LIN {X 0,Y 360.058,Z 331.263,A -85,B 0,C 180,E1 -13391.69,E2 -13391.69} C_VEL
LIN {X 0,Y 358.876,Z 343.094,A -85,B 0,C 180,E1 -13392.772,E2 -13392.772} C_VEL
LIN {X 0,Y 357.607,Z 353.882,A -85,B 0,C 180,E1 -13394.031,E2 -13394.031} C_VEL
LIN {X 0,Y 356.56,Z 363.612,A -85,B 0,C 180,E1 -13395.447,E2 -13395.447} C_VEL
LIN {X 0,Y 355.69,Z 371.607,A -85,B 0,C 180,E1 -13396.868,E2 -13396.868} C_VEL
LIN {X 0,Y 354.707,Z 379.453,A -85,B 0,C 180,E1 -13398.574,E2 -13398.574} C_VEL
LIN {X 0,Y 354.087,Z 385.752,A -85,B 0,C 180,E1 -13400.289,E2 -13400.289} C_VEL
LIN {X 0,Y 353.652,Z 390.778,A -85,B 0,C 180,E1 -13402.005,E2 -13402.005} C_VEL
LIN {X 0,Y 353.422,Z 394.956,A -85,B 0,C 180,E1 -13403.87,E2 -13403.87} C_VEL
LIN {X 0,Y 353.356,Z 397.554,A -85,B 0,C 180,E1 -13405.439,E2 -13405.439} C_VEL
LIN {X 0,Y 353.303,Z 399.885,A -85,B 0,C 180,E1 -13407.722,E2 -13407.722} C_VEL
LIN {X 0,Y 353.398,Z 400.466,A -85,B 0,C 180,E1 -13408.862,E2 -13408.862} C_VEL
LIN {X 0,Y 353.411,Z 400.609,A -85,B 0,C 180,E1 -13410.002,E2 -13410.002} C_VEL
LIN {X 0,Y 353.42,Z 400.345,A -85,B 0,C 180,E1 -13411.141,E2 -13411.141} C_VEL
LIN {X 0,Y 353.334,Z 399.683,A -85,B 0,C 180,E1 -13412.282,E2 -13412.282} C_VEL
LIN {X 0,Y 353.285,Z 398.629,A -85,B 0,C 180,E1 -13413.423,E2 -13413.423} C_VEL
LIN {X 0,Y 353.361,Z 397.134,A -85,B 0,C 180,E1 -13414.565,E2 -13414.565} C_VEL
LIN {X 0,Y 353.448,Z 394.313,A -85,B 0,C 180,E1 -13416.169,E2 -13416.169} C_VEL
LIN {X 0,Y 353.68,Z 389.954,A -85,B 0,C 180,E1 -13417.997,E2 -13417.997} C_VEL
LIN {X 0,Y 354.204,Z 383.631,A -85,B 0,C 180,E1 -13420,E2 -13420} C_VEL
LIN {X 0,Y 354.815,Z 376.746,A -85,B 0,C 180,E1 -13421.716,E2 -13421.716} C_VEL
LIN {X 0,Y 355.758,Z 368.183,A -85,B 0,C 180,E1 -13423.424,E2 -13423.424} C_VEL
LIN {X 0,Y 356.833,Z 358.104,A -85,B 0,C 180,E1 -13425.024,E2 -13425.024} C_VEL
LIN {X 0,Y 357.848,Z 347.306,A -85,B 0,C 180,E1 -13426.4,E2 -13426.4} C_VEL
LIN {X 0,Y 358.984,Z 336.101,A -85,B 0,C 180,E1 -13427.519,E2 -13427.519} C_VEL
LIN {X 0,Y 359.355,Z 329.321,A -85,B 0,C 180,E1 -13428.089,E2 -13428.089} C_VEL
LIN {X 0,Y 358.031,Z 317.342,A -85,B 0,C 180,E1 -13428.993,E2 -13428.993} C_VEL
LIN {X 0,Y 356.267,Z 304.211,A -85,B 0,C 180,E1 -13429.746,E2 -13429.746} C_VEL
LIN {X 0,Y 354.344,Z 292.6,A -85,B 0,C 180,E1 -13430.25,E2 -13430.25} C_VEL
LIN {X 0,Y 354.862,Z 285.094,A -85,B 0,C 180,E1 -13433.858,E2 -13433.858} C_VEL
LIN {X 0,Y 355.458,Z 278.242,A -85,B 0,C 180,E1 -13437.161,E2 -13437.161} C_VEL
LIN {X 0,Y 356.084,Z 272.036,A -85,B 0,C 180,E1 -13440.223,E2 -13440.223} C_VEL
LIN {X 0,Y 356.8,Z 265.53,A -85,B 0,C 180,E1 -13443.473,E2 -13443.473} C_VEL
LIN {X 0,Y 357.286,Z 260.221,A -85,B 0,C 180,E1 -13446.245,E2 -13446.245} C_VEL
LIN {X 0,Y 357.088,Z 256.908,A -85,B 0,C 180,E1 -13448.07,E2 -13448.07} C_VEL
LIN {X 0,Y 356.109,Z 251.252,A -85,B 0,C 180,E1 -13451.414,E2 -13451.414} C_VEL
LIN {X 0,Y 355.185,Z 246.213,A -85,B 0,C 180,E1 -13454.575,E2 -13454.575} C_VEL
LIN {X 0,Y 354.819,Z 244.293,A -85,B 0,C 180,E1 -13455.947,E2 -13455.947} C_VEL
LIN {X 0,Y 354.794,Z 244.292,A -85,B 0,C 180,E1 -13459.18,E2 -13459.18} C_VEL
LIN {X 0,Y 354.813,Z 244.288,A -85,B 0,C 180,E1 -13462.404,E2 -13462.404} C_VEL
LIN {X 0,Y 354.818,Z 244.287,A -85,B 0,C 180,E1 -13464.941,E2 -13464.941} C_VEL
LIN {X 0,Y 354.8,Z 244.292,A -85,B 0,C 180,E1 -13468.406,E2 -13468.406} C_VEL
LIN {X 0,Y 354.817,Z 244.284,A -85,B 0,C 180,E1 -13471.616,E2 -13471.616} C_VEL
LIN {X 0,Y 354.861,Z 244.279,A -85,B 0,C 180,E1 -13475.424,E2 -13475.424} C_VEL
LIN {X 0,Y 354.834,Z 244.282,A -85,B 0,C 180,E1 -13479.114,E2 -13479.114} C_VEL
LIN {X 0,Y 354.867,Z 244.279,A -85,B 0,C 180,E1 -13482.718,E2 -13482.718} C_VEL
LIN {X 0,Y 354.947,Z 244.271,A -85,B 0,C 180,E1 -13486.255,E2 -13486.255} C_VEL
LIN {X 0,Y 354.959,Z 244.272,A -85,B 0,C 180,E1 -13489.735,E2 -13489.735} C_VEL
LIN {X 0,Y 355.117,Z 244.248,A -85,B 0,C 180,E1 -13493.18,E2 -13493.18} C_VEL
LIN {X 0,Y 355.251,Z 244.235,A -85,B 0,C 180,E1 -13497.733,E2 -13497.733} C_VEL
LIN {X 0,Y 355.36,Z 244.218,A -85,B 0,C 180,E1 -13500,E2 -13500} C_VEL
LIN {X 0,Y 355.24,Z 244.232,A -85,B 0,C 180,E1 -13502.268,E2 -13502.268} C_VEL
LIN {X 0,Y 355.09,Z 244.252,A -85,B 0,C 180,E1 -13506.82,E2 -13506.82} C_VEL
LIN {X 0,Y 354.962,Z 244.266,A -85,B 0,C 180,E1 -13510.265,E2 -13510.265} C_VEL
LIN {X 0,Y 354.951,Z 244.267,A -85,B 0,C 180,E1 -13514.019,E2 -13514.019} C_VEL
LIN {X 0,Y 354.898,Z 244.274,A -85,B 0,C 180,E1 -13518.092,E2 -13518.092} C_VEL
LIN {X 0,Y 354.821,Z 244.284,A -85,B 0,C 180,E1 -13522.107,E2 -13522.107} C_VEL
LIN {X 0,Y 354.806,Z 244.286,A -85,B 0,C 180,E1 -13525.835,E2 -13525.835} C_VEL
LIN {X 0,Y 354.804,Z 244.286,A -85,B 0,C 180,E1 -13529.683,E2 -13529.683} C_VEL
LIN {X 0,Y 354.795,Z 244.291,A -85,B 0,C 180,E1 -13532.333,E2 -13532.333} C_VEL
LIN {X 0,Y 354.829,Z 244.283,A -85,B 0,C 180,E1 -13535.699,E2 -13535.699} C_VEL
LIN {X 0,Y 354.832,Z 244.282,A -85,B 0,C 180,E1 -13539.423,E2 -13539.423} C_VEL
LIN {X 0,Y 354.795,Z 244.288,A -85,B 0,C 180,E1 -13542.866,E2 -13542.866} C_VEL
LIN {X 0,Y 354.77,Z 244.296,A -85,B 0,C 180,E1 -13546.102,E2 -13546.102} C_VEL
LIN {X 0,Y 354.769,Z 244.29,A -85,B 0,C 180,E1 -13549.175,E2 -13549.175} C_VEL
LIN {X 0,Y 354.806,Z 244.287,A -85,B 0,C 180,E1 -13552.403,E2 -13552.403} C_VEL
LIN {X 0,Y 354.813,Z 244.285,A -85,B 0,C 180,E1 -13554.939,E2 -13554.939} C_VEL
LIN {X 0,Y 354.704,Z 244.299,A -85,B 0,C 180,E1 -13558.429,E2 -13558.429} C_VEL
LIN {X 0,Y 354.372,Z 244.344,A -85,B 0,C 180,E1 -13561.576,E2 -13561.576} C_VEL
LIN {X 0,Y 354.235,Z 244.363,A -85,B 0,C 180,E1 -13562.849,E2 -13562.849} C_VEL
LIN {X 0,Y 354.103,Z 247.731,A -85,B 0,C 180,E1 -13566.611,E2 -13566.611} C_VEL
LIN {X 0,Y 353.973,Z 251.128,A -85,B 0,C 180,E1 -13570.272,E2 -13570.272} C_VEL
LIN {X 0,Y 353.975,Z 253.452,A -85,B 0,C 180,E1 -13572.672,E2 -13572.672} C_VEL
LIN {X 0,Y 353.925,Z 254.896,A -85,B 0,C 180,E1 -13574.115,E2 -13574.115} C_VEL
LIN {X 0,Y 357.65,Z 268.629,A -85,B 0,C 180,E1 -13574.87,E2 -13574.87} C_VEL
LIN {X 0,Y 360.102,Z 279.83,A -85,B 0,C 180,E1 -13575.653,E2 -13575.653} C_VEL
LIN {X 0,Y 360.581,Z 283.09,A -85,B 0,C 180,E1 -13575.906,E2 -13575.906} C_VEL
LIN {X 0,Y 359.816,Z 293.602,A -85,B 0,C 180,E1 -13576.731,E2 -13576.731} C_VEL
LIN {X 0,Y 358.891,Z 304.794,A -85,B 0,C 180,E1 -13577.846,E2 -13577.846} C_VEL
LIN {X 0,Y 357.921,Z 315.075,A -85,B 0,C 180,E1 -13579.131,E2 -13579.131} C_VEL
LIN {X 0,Y 356.846,Z 324.774,A -85,B 0,C 180,E1 -13580.647,E2 -13580.647} C_VEL
LIN {X 0,Y 355.979,Z 333.461,A -85,B 0,C 180,E1 -13582.34,E2 -13582.34} C_VEL
LIN {X 0,Y 355.2,Z 340.428,A -85,B 0,C 180,E1 -13584.036,E2 -13584.036} C_VEL
LIN {X 0,Y 354.497,Z 345.168,A -85,B 0,C 180,E1 -13585.45,E2 -13585.45} C_VEL
LIN {X 0,Y 354.096,Z 349.736,A -85,B 0,C 180,E1 -13587.154,E2 -13587.154} C_VEL
LIN {X 0,Y 353.696,Z 353.231,A -85,B 0,C 180,E1 -13588.86,E2 -13588.86} C_VEL
LIN {X 0,Y 353.581,Z 355.01,A -85,B 0,C 180,E1 -13589.998,E2 -13589.998} C_VEL
LIN {X 0,Y 353.583,Z 357.296,A -85,B 0,C 180,E1 -13592.277,E2 -13592.277} C_VEL
LIN {X 0,Y 353.509,Z 357.876,A -85,B 0,C 180,E1 -13593.418,E2 -13593.418} C_VEL
LIN {X 0,Y 353.499,Z 358.05,A -85,B 0,C 180,E1 -13594.56,E2 -13594.56} C_VEL
LIN {X 0,Y 353.625,Z 357.48,A -85,B 0,C 180,E1 -13596.427,E2 -13596.427} C_VEL
LIN {X 0,Y 353.735,Z 356.197,A -85,B 0,C 180,E1 -13597.993,E2 -13597.993} C_VEL
LIN {X 0,Y 353.889,Z 354.775,A -85,B 0,C 180,E1 -13599.14,E2 -13599.14} C_VEL
LIN {X 0,Y 354.259,Z 351.838,A -85,B 0,C 180,E1 -13600.862,E2 -13600.862} C_VEL
LIN {X 0,Y 354.817,Z 347.848,A -85,B 0,C 180,E1 -13602.583,E2 -13602.583} C_VEL
LIN {X 0,Y 355.547,Z 342.349,A -85,B 0,C 180,E1 -13604.401,E2 -13604.401} C_VEL
LIN {X 0,Y 356.574,Z 334.948,A -85,B 0,C 180,E1 -13606.31,E2 -13606.31} C_VEL
LIN {X 0,Y 357.752,Z 326.529,A -85,B 0,C 180,E1 -13608.022,E2 -13608.022} C_VEL
LIN {X 0,Y 358.863,Z 317.829,A -85,B 0,C 180,E1 -13609.445,E2 -13609.445} C_VEL
LIN {X 0,Y 359.9,Z 308.259,A -85,B 0,C 180,E1 -13610.726,E2 -13610.726} C_VEL
LIN {X 0,Y 361.08,Z 297.77,A -85,B 0,C 180,E1 -13611.852,E2 -13611.852} C_VEL
LIN {X 0,Y 362.032,Z 286.148,A -85,B 0,C 180,E1 -13612.844,E2 -13612.844} C_VEL
LIN {X 0,Y 361.97,Z 283.598,A -85,B 0,C 180,E1 -13613.04,E2 -13613.04} C_VEL
LIN {X 0,Y 359.075,Z 271.49,A -85,B 0,C 180,E1 -13614.013,E2 -13614.013} C_VEL
LIN {X 0,Y 355.266,Z 259.208,A -85,B 0,C 180,E1 -13614.823,E2 -13614.823} C_VEL
LIN {X 0,Y 354.079,Z 255.183,A -85,B 0,C 180,E1 -13615.056,E2 -13615.056} C_VEL
LIN {X 0,Y 354.18,Z 252.024,A -85,B 0,C 180,E1 -13618.437,E2 -13618.437} C_VEL
LIN {X 0,Y 354.315,Z 248.516,A -85,B 0,C 180,E1 -13622.379,E2 -13622.379} C_VEL
LIN {X 0,Y 354.434,Z 245.746,A -85,B 0,C 180,E1 -13625.611,E2 -13625.611} C_VEL
LIN {X 0,Y 354.548,Z 244.323,A -85,B 0,C 180,E1 -13627.542,E2 -13627.542} C_VEL
LIN {X 0,Y 354.58,Z 244.316,A -85,B 0,C 180,E1 -13628.172,E2 -13628.172} C_VEL
LIN {X 0,Y 353.94,Z 244.397,A -85,B 0,C 180,E1 -13629.122,E2 -13629.122} C_VEL
LIN {X 0,Y 351.13,Z 244.747,A -85,B 0,C 180,E1 -13630.667,E2 -13630.667} C_VEL
LIN {X 0,Y 348.761,Z 245.041,A -85,B 0,C 180,E1 -13631.917,E2 -13631.917} C_VEL
LIN {X 0,Y 347.775,Z 245.167,A -85,B 0,C 180,E1 -13632.884,E2 -13632.884} C_VEL
LIN {X 0,Y 347.711,Z 245.172,A -85,B 0,C 180,E1 -13633.211,E2 -13633.211} C_VEL
LIN {X 0,Y 347.718,Z 245.172,A -85,B 0,C 180,E1 -13636.685,E2 -13636.685} C_VEL
LIN {X 0,Y 347.739,Z 245.169,A -85,B 0,C 180,E1 -13640.172,E2 -13640.172} C_VEL
LIN {X 0,Y 347.757,Z 245.167,A -85,B 0,C 180,E1 -13642.678,E2 -13642.678} C_VEL
LIN {X 0,Y 347.739,Z 245.168,A -85,B 0,C 180,E1 -13645.955,E2 -13645.955} C_VEL
LIN {X 0,Y 347.74,Z 245.168,A -85,B 0,C 180,E1 -13649.651,E2 -13649.651} C_VEL
LIN {X 0,Y 347.821,Z 245.157,A -85,B 0,C 180,E1 -13653.607,E2 -13653.607} C_VEL
LIN {X 0,Y 347.778,Z 245.165,A -85,B 0,C 180,E1 -13656.161,E2 -13656.161} C_VEL
LIN {X 0,Y 347.802,Z 245.16,A -85,B 0,C 180,E1 -13659.908,E2 -13659.908} C_VEL
LIN {X 0,Y 347.855,Z 245.156,A -85,B 0,C 180,E1 -13662.358,E2 -13662.358} C_VEL
LIN {X 0,Y 347.886,Z 245.15,A -85,B 0,C 180,E1 -13665.97,E2 -13665.97} C_VEL
LIN {X 0,Y 347.917,Z 245.147,A -85,B 0,C 180,E1 -13669.525,E2 -13669.525} C_VEL
LIN {X 0,Y 348.1,Z 245.122,A -85,B 0,C 180,E1 -13673.042,E2 -13673.042} C_VEL
LIN {X 0,Y 348.198,Z 245.111,A -85,B 0,C 180,E1 -13677.686,E2 -13677.686} C_VEL
LIN {X 0,Y 348.313,Z 245.098,A -85,B 0,C 180,E1 -13680,E2 -13680} C_VEL
LIN {X 0,Y 348.197,Z 245.113,A -85,B 0,C 180,E1 -13682.313,E2 -13682.313} C_VEL
LIN {X 0,Y 348.1,Z 245.125,A -85,B 0,C 180,E1 -13686.958,E2 -13686.958} C_VEL
LIN {X 0,Y 347.917,Z 245.147,A -85,B 0,C 180,E1 -13690.475,E2 -13690.475} C_VEL
LIN {X 0,Y 347.887,Z 245.149,A -85,B 0,C 180,E1 -13694.15,E2 -13694.15} C_VEL
LIN {X 0,Y 347.88,Z 245.151,A -85,B 0,C 180,E1 -13698.291,E2 -13698.291} C_VEL
LIN {X 0,Y 347.778,Z 245.165,A -85,B 0,C 180,E1 -13701.636,E2 -13701.636} C_VEL
LIN {X 0,Y 347.802,Z 245.164,A -85,B 0,C 180,E1 -13705.109,E2 -13705.109} C_VEL
LIN {X 0,Y 347.802,Z 245.161,A -85,B 0,C 180,E1 -13707.695,E2 -13707.695} C_VEL
LIN {X 0,Y 347.76,Z 245.169,A -85,B 0,C 180,E1 -13710.347,E2 -13710.347} C_VEL
LIN {X 0,Y 347.738,Z 245.17,A -85,B 0,C 180,E1 -13714.045,E2 -13714.045} C_VEL
LIN {X 0,Y 347.752,Z 245.165,A -85,B 0,C 180,E1 -13717.322,E2 -13717.322} C_VEL
LIN {X 0,Y 347.723,Z 245.173,A -85,B 0,C 180,E1 -13720.298,E2 -13720.298} C_VEL
LIN {X 0,Y 347.768,Z 245.367,A -85,B 0,C 180,E1 -13722.022,E2 -13722.022} C_VEL
LIN {X 0,Y 348.571,Z 249.606,A -85,B 0,C 180,E1 -13725.118,E2 -13725.118} C_VEL
LIN {X 0,Y 349.498,Z 254.495,A -85,B 0,C 180,E1 -13728.428,E2 -13728.428} C_VEL
LIN {X 0,Y 350.331,Z 259.441,A -85,B 0,C 180,E1 -13731.548,E2 -13731.548} C_VEL
LIN {X 0,Y 350.61,Z 262.393,A -85,B 0,C 180,E1 -13733.303,E2 -13733.303} C_VEL
LIN {X 0,Y 350.176,Z 266.899,A -85,B 0,C 180,E1 -13735.811,E2 -13735.811} C_VEL
LIN {X 0,Y 349.329,Z 273.141,A -85,B 0,C 180,E1 -13739.137,E2 -13739.137} C_VEL
LIN {X 0,Y 348.626,Z 279.606,A -85,B 0,C 180,E1 -13742.499,E2 -13742.499} C_VEL
LIN {X 0,Y 347.841,Z 286.858,A -85,B 0,C 180,E1 -13746.168,E2 -13746.168} C_VEL
LIN {X 0,Y 347.476,Z 292.026,A -85,B 0,C 180,E1 -13748.76,E2 -13748.76} C_VEL
LIN {X 0,Y 350.202,Z 305.797,A -85,B 0,C 180,E1 -13749.447,E2 -13749.447} C_VEL
LIN {X 0,Y 351.954,Z 318.039,A -85,B 0,C 180,E1 -13750.244,E2 -13750.244} C_VEL
LIN {X 0,Y 353.126,Z 331.267,A -85,B 0,C 180,E1 -13751.322,E2 -13751.322} C_VEL
LIN {X 0,Y 352.574,Z 338.737,A -85,B 0,C 180,E1 -13752.005,E2 -13752.005} C_VEL
LIN {X 0,Y 351.173,Z 350.363,A -85,B 0,C 180,E1 -13753.282,E2 -13753.282} C_VEL
LIN {X 0,Y 349.953,Z 360.339,A -85,B 0,C 180,E1 -13754.662,E2 -13754.662} C_VEL
LIN {X 0,Y 348.939,Z 369.84,A -85,B 0,C 180,E1 -13756.312,E2 -13756.312} C_VEL
LIN {X 0,Y 347.863,Z 377.945,A -85,B 0,C 180,E1 -13758.05,E2 -13758.05} C_VEL
LIN {X 0,Y 347.288,Z 383.468,A -85,B 0,C 180,E1 -13759.508,E2 -13759.508} C_VEL
LIN {X 0,Y 346.737,Z 388.884,A -85,B 0,C 180,E1 -13761.258,E2 -13761.258} C_VEL
LIN {X 0,Y 346.418,Z 393.127,A -85,B 0,C 180,E1 -13763.01,E2 -13763.01} C_VEL
LIN {X 0,Y 346.317,Z 395.385,A -85,B 0,C 180,E1 -13764.178,E2 -13764.178} C_VEL
LIN {X 0,Y 346.27,Z 397.163,A -85,B 0,C 180,E1 -13765.345,E2 -13765.345} C_VEL
LIN {X 0,Y 346.208,Z 399.478,A -85,B 0,C 180,E1 -13767.675,E2 -13767.675} C_VEL
LIN {X 0,Y 346.318,Z 400.049,A -85,B 0,C 180,E1 -13768.839,E2 -13768.839} C_VEL
LIN {X 0,Y 346.35,Z 400.179,A -85,B 0,C 180,E1 -13770.002,E2 -13770.002} C_VEL
LIN {X 0,Y 346.339,Z 399.906,A -85,B 0,C 180,E1 -13771.164,E2 -13771.164} C_VEL
LIN {X 0,Y 346.207,Z 398.173,A -85,B 0,C 180,E1 -13773.493,E2 -13773.493} C_VEL
LIN {X 0,Y 346.275,Z 396.66,A -85,B 0,C 180,E1 -13774.658,E2 -13774.658} C_VEL
LIN {X 0,Y 346.347,Z 394.16,A -85,B 0,C 180,E1 -13776.12,E2 -13776.12} C_VEL
LIN {X 0,Y 346.61,Z 389.441,A -85,B 0,C 180,E1 -13778.161,E2 -13778.161} C_VEL
LIN {X 0,Y 347.17,Z 383.096,A -85,B 0,C 180,E1 -13780.204,E2 -13780.204} C_VEL
LIN {X 0,Y 347.826,Z 376.188,A -85,B 0,C 180,E1 -13781.954,E2 -13781.954} C_VEL
LIN {X 0,Y 348.665,Z 369.151,A -85,B 0,C 180,E1 -13783.405,E2 -13783.405} C_VEL
LIN {X 0,Y 349.601,Z 360.673,A -85,B 0,C 180,E1 -13784.853,E2 -13784.853} C_VEL
LIN {X 0,Y 350.656,Z 350.206,A -85,B 0,C 180,E1 -13786.297,E2 -13786.297} C_VEL
LIN {X 0,Y 351.726,Z 339.857,A -85,B 0,C 180,E1 -13787.443,E2 -13787.443} C_VEL
LIN {X 0,Y 352.464,Z 330.296,A -85,B 0,C 180,E1 -13788.305,E2 -13788.305} C_VEL
LIN {X 0,Y 351.097,Z 317.439,A -85,B 0,C 180,E1 -13789.314,E2 -13789.314} C_VEL
LIN {X 0,Y 349.341,Z 304.374,A -85,B 0,C 180,E1 -13790.094,E2 -13790.094} C_VEL
LIN {X 0,Y 347.302,Z 292.128,A -85,B 0,C 180,E1 -13790.664,E2 -13790.664} C_VEL
LIN {X 0,Y 347.899,Z 284.112,A -85,B 0,C 180,E1 -13794.624,E2 -13794.624} C_VEL
LIN {X 0,Y 348.652,Z 276.76,A -85,B 0,C 180,E1 -13798.277,E2 -13798.277} C_VEL
LIN {X 0,Y 349.573,Z 268.667,A -85,B 0,C 180,E1 -13802.393,E2 -13802.393} C_VEL
LIN {X 0,Y 350.24,Z 262.592,A -85,B 0,C 180,E1 -13805.588,E2 -13805.588} C_VEL
LIN {X 0,Y 350.162,Z 258.748,A -85,B 0,C 180,E1 -13807.722,E2 -13807.722} C_VEL
LIN {X 0,Y 349.3,Z 253.492,A -85,B 0,C 180,E1 -13810.838,E2 -13810.838} C_VEL
LIN {X 0,Y 348.31,Z 248.14,A -85,B 0,C 180,E1 -13814.251,E2 -13814.251} C_VEL
LIN {X 0,Y 347.737,Z 245.175,A -85,B 0,C 180,E1 -13816.294,E2 -13816.294} C_VEL
LIN {X 0,Y 347.739,Z 245.172,A -85,B 0,C 180,E1 -13819.704,E2 -13819.704} C_VEL
LIN {X 0,Y 347.768,Z 245.168,A -85,B 0,C 180,E1 -13822.68,E2 -13822.68} C_VEL
LIN {X 0,Y 347.755,Z 245.165,A -85,B 0,C 180,E1 -13825.957,E2 -13825.957} C_VEL
LIN {X 0,Y 347.749,Z 245.165,A -85,B 0,C 180,E1 -13829.652,E2 -13829.652} C_VEL
LIN {X 0,Y 347.791,Z 245.16,A -85,B 0,C 180,E1 -13833.604,E2 -13833.604} C_VEL
LIN {X 0,Y 347.793,Z 245.165,A -85,B 0,C 180,E1 -13836.162,E2 -13836.162} C_VEL
LIN {X 0,Y 347.803,Z 245.162,A -85,B 0,C 180,E1 -13839.909,E2 -13839.909} C_VEL
LIN {X 0,Y 347.84,Z 245.156,A -85,B 0,C 180,E1 -13842.358,E2 -13842.358} C_VEL
LIN {X 0,Y 347.906,Z 245.151,A -85,B 0,C 180,E1 -13845.971,E2 -13845.971} C_VEL
LIN {X 0,Y 347.899,Z 245.149,A -85,B 0,C 180,E1 -13849.525,E2 -13849.525} C_VEL
LIN {X 0,Y 348.084,Z 245.123,A -85,B 0,C 180,E1 -13853.042,E2 -13853.042} C_VEL
LIN {X 0,Y 348.213,Z 245.112,A -85,B 0,C 180,E1 -13857.687,E2 -13857.687} C_VEL
LIN {X 0,Y 348.311,Z 245.096,A -85,B 0,C 180,E1 -13860,E2 -13860} C_VEL
LIN {X 0,Y 348.202,Z 245.108,A -85,B 0,C 180,E1 -13862.314,E2 -13862.314} C_VEL
LIN {X 0,Y 348.058,Z 245.129,A -85,B 0,C 180,E1 -13866.959,E2 -13866.959} C_VEL
LIN {X 0,Y 347.902,Z 245.146,A -85,B 0,C 180,E1 -13870.475,E2 -13870.475} C_VEL
LIN {X 0,Y 347.907,Z 245.145,A -85,B 0,C 180,E1 -13874.15,E2 -13874.15} C_VEL
LIN {X 0,Y 347.837,Z 245.154,A -85,B 0,C 180,E1 -13878.259,E2 -13878.259} C_VEL
LIN {X 0,Y 347.775,Z 245.162,A -85,B 0,C 180,E1 -13881.625,E2 -13881.625} C_VEL
LIN {X 0,Y 347.744,Z 245.168,A -85,B 0,C 180,E1 -13885.114,E2 -13885.114} C_VEL
LIN {X 0,Y 347.735,Z 245.166,A -85,B 0,C 180,E1 -13887.701,E2 -13887.701} C_VEL
LIN {X 0,Y 347.746,Z 245.168,A -85,B 0,C 180,E1 -13890.349,E2 -13890.349} C_VEL
LIN {X 0,Y 347.756,Z 245.165,A -85,B 0,C 180,E1 -13894.043,E2 -13894.043} C_VEL
LIN {X 0,Y 347.768,Z 245.162,A -85,B 0,C 180,E1 -13897.32,E2 -13897.32} C_VEL
LIN {X 0,Y 347.739,Z 245.172,A -85,B 0,C 180,E1 -13900.296,E2 -13900.296} C_VEL
LIN {X 0,Y 347.73,Z 245.167,A -85,B 0,C 180,E1 -13903.407,E2 -13903.407} C_VEL
LIN {X 0,Y 347.729,Z 245.168,A -85,B 0,C 180,E1 -13906.686,E2 -13906.686} C_VEL
LIN {X 0,Y 347.707,Z 245.174,A -85,B 0,C 180,E1 -13910.182,E2 -13910.182} C_VEL
LIN {X 0,Y 347.762,Z 245.164,A -85,B 0,C 180,E1 -13912.677,E2 -13912.677} C_VEL
LIN {X 0,Y 347.754,Z 245.169,A -85,B 0,C 180,E1 -13915.955,E2 -13915.955} C_VEL
LIN {X 0,Y 347.669,Z 245.176,A -85,B 0,C 180,E1 -13918.291,E2 -13918.291} C_VEL
LIN {X 0,Y 347.404,Z 245.208,A -85,B 0,C 180,E1 -13920.952,E2 -13920.952} C_VEL
LIN {X 0,Y 347.201,Z 245.357,A -85,B 0,C 180,E1 -13922.955,E2 -13922.955} C_VEL
LIN {X 0,Y 347.086,Z 248.146,A -85,B 0,C 180,E1 -13926.109,E2 -13926.109} C_VEL
LIN {X 0,Y 346.925,Z 251.58,A -85,B 0,C 180,E1 -13929.854,E2 -13929.854} C_VEL
LIN {X 0,Y 346.926,Z 253.929,A -85,B 0,C 180,E1 -13932.308,E2 -13932.308} C_VEL
LIN {X 0,Y 346.884,Z 255.292,A -85,B 0,C 180,E1 -13933.706,E2 -13933.706} C_VEL
LIN {X 0,Y 350.877,Z 270.053,A -85,B 0,C 180,E1 -13934.567,E2 -13934.567} C_VEL
LIN {X 0,Y 353.586,Z 282.574,A -85,B 0,C 180,E1 -13935.495,E2 -13935.495} C_VEL
LIN {X 0,Y 353.542,Z 287.207,A -85,B 0,C 180,E1 -13935.846,E2 -13935.846} C_VEL
LIN {X 0,Y 352.538,Z 299.056,A -85,B 0,C 180,E1 -13936.892,E2 -13936.892} C_VEL
LIN {X 0,Y 351.567,Z 310.381,A -85,B 0,C 180,E1 -13938.175,E2 -13938.175} C_VEL
LIN {X 0,Y 350.442,Z 320.404,A -85,B 0,C 180,E1 -13939.6,E2 -13939.6} C_VEL
LIN {X 0,Y 349.566,Z 328.577,A -85,B 0,C 180,E1 -13941.034,E2 -13941.034} C_VEL
LIN {X 0,Y 348.699,Z 336.58,A -85,B 0,C 180,E1 -13942.762,E2 -13942.762} C_VEL
LIN {X 0,Y 348.028,Z 342.031,A -85,B 0,C 180,E1 -13944.203,E2 -13944.203} C_VEL
LIN {X 0,Y 347.333,Z 347.366,A -85,B 0,C 180,E1 -13945.937,E2 -13945.937} C_VEL
LIN {X 0,Y 346.814,Z 351.54,A -85,B 0,C 180,E1 -13947.676,E2 -13947.676} C_VEL
LIN {X 0,Y 346.626,Z 353.752,A -85,B 0,C 180,E1 -13948.837,E2 -13948.837} C_VEL
LIN {X 0,Y 346.511,Z 355.5,A -85,B 0,C 180,E1 -13949.998,E2 -13949.998} C_VEL
LIN {X 0,Y 346.502,Z 357.758,A -85,B 0,C 180,E1 -13952.323,E2 -13952.323} C_VEL
LIN {X 0,Y 346.418,Z 358.325,A -85,B 0,C 180,E1 -13953.488,E2 -13953.488} C_VEL
LIN {X 0,Y 346.434,Z 358.47,A -85,B 0,C 180,E1 -13954.653,E2 -13954.653} C_VEL
LIN {X 0,Y 346.554,Z 357.958,A -85,B 0,C 180,E1 -13956.429,E2 -13956.429} C_VEL
LIN {X 0,Y 346.685,Z 356.574,A -85,B 0,C 180,E1 -13958.156,E2 -13958.156} C_VEL
LIN {X 0,Y 346.846,Z 355.124,A -85,B 0,C 180,E1 -13959.327,E2 -13959.327} C_VEL
LIN {X 0,Y 347.234,Z 352.157,A -85,B 0,C 180,E1 -13961.084,E2 -13961.084} C_VEL
LIN {X 0,Y 347.834,Z 348.133,A -85,B 0,C 180,E1 -13962.84,E2 -13962.84} C_VEL
LIN {X 0,Y 348.739,Z 341.951,A -85,B 0,C 180,E1 -13964.881,E2 -13964.881} C_VEL
LIN {X 0,Y 349.732,Z 335.154,A -85,B 0,C 180,E1 -13966.638,E2 -13966.638} C_VEL
LIN {X 0,Y 350.935,Z 326.664,A -85,B 0,C 180,E1 -13968.384,E2 -13968.384} C_VEL
LIN {X 0,Y 352.249,Z 316.602,A -85,B 0,C 180,E1 -13970.028,E2 -13970.028} C_VEL
LIN {X 0,Y 353.393,Z 307.088,A -85,B 0,C 180,E1 -13971.279,E2 -13971.279} C_VEL
LIN {X 0,Y 354.626,Z 296.163,A -85,B 0,C 180,E1 -13972.424,E2 -13972.424} C_VEL
LIN {X 0,Y 355.417,Z 285.856,A -85,B 0,C 180,E1 -13973.294,E2 -13973.294} C_VEL
LIN {X 0,Y 352.732,Z 274.226,A -85,B 0,C 180,E1 -13974.28,E2 -13974.28} C_VEL
LIN {X 0,Y 348.994,Z 261.751,A -85,B 0,C 180,E1 -13975.164,E2 -13975.164} C_VEL
LIN {X 0,Y 347.031,Z 255.628,A -85,B 0,C 180,E1 -13975.529,E2 -13975.529} C_VEL
LIN {X 0,Y 347.181,Z 252.009,A -85,B 0,C 180,E1 -13979.488,E2 -13979.488} C_VEL
LIN {X 0,Y 347.319,Z 248.849,A -85,B 0,C 180,E1 -13983.114,E2 -13983.114} C_VEL
LIN {X 0,Y 347.426,Z 246.418,A -85,B 0,C 180,E1 -13985.986,E2 -13985.986} C_VEL
LIN {X 0,Y 347.477,Z 245.306,A -85,B 0,C 180,E1 -13987.354,E2 -13987.354} C_VEL
LIN {X 0,Y 347.656,Z 245.178,A -85,B 0,C 180,E1 -13990.305,E2 -13990.305} C_VEL
LIN {X 0,Y 347.711,Z 245.172,A -85,B 0,C 180,E1 -13993.211,E2 -13993.211} C_VEL
LIN {X 0,Y 347.09,Z 245.256,A -85,B 0,C 180,E1 -13994.178,E2 -13994.178} C_VEL
LIN {X 0,Y 344.251,Z 245.612,A -85,B 0,C 180,E1 -13995.75,E2 -13995.75} C_VEL
LIN {X 0,Y 341.815,Z 245.911,A -85,B 0,C 180,E1 -13997.023,E2 -13997.023} C_VEL
LIN {X 0,Y 340.764,Z 246.04,A -85,B 0,C 180,E1 -13998.009,E2 -13998.009} C_VEL
LIN {X 0,Y 340.677,Z 246.049,A -85,B 0,C 180,E1 -13998.342,E2 -13998.342} C_VEL
LIN {X 0,Y 340.727,Z 246.042,A -85,B 0,C 180,E1 -14001.771,E2 -14001.771} C_VEL
LIN {X 0,Y 340.714,Z 246.045,A -85,B 0,C 180,E1 -14005.594,E2 -14005.594} C_VEL
LIN {X 0,Y 340.688,Z 246.046,A -85,B 0,C 180,E1 -14008.954,E2 -14008.954} C_VEL
LIN {X 0,Y 340.793,Z 246.032,A -85,B 0,C 180,E1 -14013.019,E2 -14013.019} C_VEL
LIN {X 0,Y 340.746,Z 246.041,A -85,B 0,C 180,E1 -14015.637,E2 -14015.637} C_VEL
LIN {X 0,Y 340.742,Z 246.041,A -85,B 0,C 180,E1 -14019.474,E2 -14019.474} C_VEL
LIN {X 0,Y 340.847,Z 246.027,A -85,B 0,C 180,E1 -14021.983,E2 -14021.983} C_VEL
LIN {X 0,Y 340.858,Z 246.027,A -85,B 0,C 180,E1 -14025.704,E2 -14025.704} C_VEL
LIN {X 0,Y 340.859,Z 246.027,A -85,B 0,C 180,E1 -14029.306,E2 -14029.306} C_VEL
LIN {X 0,Y 341.069,Z 245.998,A -85,B 0,C 180,E1 -14032.898,E2 -14032.898} C_VEL
LIN {X 0,Y 341.16,Z 245.988,A -85,B 0,C 180,E1 -14037.639,E2 -14037.639} C_VEL
LIN {X 0,Y 341.263,Z 245.976,A -85,B 0,C 180,E1 -14040,E2 -14040} C_VEL
LIN {X 0,Y 341.159,Z 245.99,A -85,B 0,C 180,E1 -14042.361,E2 -14042.361} C_VEL
LIN {X 0,Y 341.069,Z 246.001,A -85,B 0,C 180,E1 -14047.102,E2 -14047.102} C_VEL
LIN {X 0,Y 340.859,Z 246.026,A -85,B 0,C 180,E1 -14050.694,E2 -14050.694} C_VEL
LIN {X 0,Y 340.851,Z 246.025,A -85,B 0,C 180,E1 -14054.325,E2 -14054.325} C_VEL
LIN {X 0,Y 340.827,Z 246.028,A -85,B 0,C 180,E1 -14058.467,E2 -14058.467} C_VEL
LIN {X 0,Y 340.743,Z 246.042,A -85,B 0,C 180,E1 -14061.858,E2 -14061.858} C_VEL
LIN {X 0,Y 340.762,Z 246.038,A -85,B 0,C 180,E1 -14065.665,E2 -14065.665} C_VEL
LIN {X 0,Y 340.732,Z 246.043,A -85,B 0,C 180,E1 -14068.32,E2 -14068.32} C_VEL
LIN {X 0,Y 340.706,Z 246.045,A -85,B 0,C 180,E1 -14071.044,E2 -14071.044} C_VEL
LIN {X 0,Y 340.708,Z 246.042,A -85,B 0,C 180,E1 -14075.28,E2 -14075.28} C_VEL
LIN {X 0,Y 340.701,Z 246.049,A -85,B 0,C 180,E1 -14078.387,E2 -14078.387} C_VEL
LIN {X 0,Y 340.678,Z 246.053,A -85,B 0,C 180,E1 -14081.311,E2 -14081.311} C_VEL
LIN {X 0,Y 341.462,Z 250.14,A -85,B 0,C 180,E1 -14084.41,E2 -14084.41} C_VEL
LIN {X 0,Y 342.525,Z 255.758,A -85,B 0,C 180,E1 -14088.328,E2 -14088.328} C_VEL
LIN {X 0,Y 343.264,Z 260.001,A -85,B 0,C 180,E1 -14091.079,E2 -14091.079} C_VEL
LIN {X 0,Y 343.625,Z 262.974,A -85,B 0,C 180,E1 -14092.906,E2 -14092.906} C_VEL
LIN {X 0,Y 343.184,Z 267.901,A -85,B 0,C 180,E1 -14095.727,E2 -14095.727} C_VEL
LIN {X 0,Y 342.168,Z 275.04,A -85,B 0,C 180,E1 -14099.617,E2 -14099.617} C_VEL
LIN {X 0,Y 341.433,Z 281.569,A -85,B 0,C 180,E1 -14103.076,E2 -14103.076} C_VEL
LIN {X 0,Y 340.653,Z 288.993,A -85,B 0,C 180,E1 -14106.924,E2 -14106.924} C_VEL
LIN {X 0,Y 340.461,Z 291.654,A -85,B 0,C 180,E1 -14108.267,E2 -14108.267} C_VEL
LIN {X 0,Y 343.237,Z 305.039,A -85,B 0,C 180,E1 -14108.958,E2 -14108.958} C_VEL
LIN {X 0,Y 344.98,Z 316.842,A -85,B 0,C 180,E1 -14109.739,E2 -14109.739} C_VEL
LIN {X 0,Y 346.149,Z 330.017,A -85,B 0,C 180,E1 -14110.825,E2 -14110.825} C_VEL
LIN {X 0,Y 346.177,Z 335.646,A -85,B 0,C 180,E1 -14111.354,E2 -14111.354} C_VEL
LIN {X 0,Y 344.814,Z 346.659,A -85,B 0,C 180,E1 -14112.506,E2 -14112.506} C_VEL
LIN {X 0,Y 343.514,Z 356.894,A -85,B 0,C 180,E1 -14113.862,E2 -14113.862} C_VEL
LIN {X 0,Y 342.333,Z 366.469,A -85,B 0,C 180,E1 -14115.436,E2 -14115.436} C_VEL
LIN {X 0,Y 341.418,Z 373.826,A -85,B 0,C 180,E1 -14116.915,E2 -14116.915} C_VEL
LIN {X 0,Y 340.447,Z 381.082,A -85,B 0,C 180,E1 -14118.692,E2 -14118.692} C_VEL
LIN {X 0,Y 339.847,Z 386.902,A -85,B 0,C 180,E1 -14120.479,E2 -14120.479} C_VEL
LIN {X 0,Y 339.416,Z 391.498,A -85,B 0,C 180,E1 -14122.267,E2 -14122.267} C_VEL
LIN {X 0,Y 339.237,Z 395.009,A -85,B 0,C 180,E1 -14124.056,E2 -14124.056} C_VEL
LIN {X 0,Y 339.188,Z 396.773,A -85,B 0,C 180,E1 -14125.248,E2 -14125.248} C_VEL
LIN {X 0,Y 339.128,Z 398.119,A -85,B 0,C 180,E1 -14126.437,E2 -14126.437} C_VEL
LIN {X 0,Y 339.223,Z 399.631,A -85,B 0,C 180,E1 -14128.815,E2 -14128.815} C_VEL
LIN {X 0,Y 339.29,Z 399.75,A -85,B 0,C 180,E1 -14130.002,E2 -14130.002} C_VEL
LIN {X 0,Y 339.26,Z 399.467,A -85,B 0,C 180,E1 -14131.189,E2 -14131.189} C_VEL
LIN {X 0,Y 339.132,Z 397.714,A -85,B 0,C 180,E1 -14133.566,E2 -14133.566} C_VEL
LIN {X 0,Y 339.194,Z 396.185,A -85,B 0,C 180,E1 -14134.756,E2 -14134.756} C_VEL
LIN {X 0,Y 339.3,Z 393.091,A -85,B 0,C 180,E1 -14136.543,E2 -14136.543} C_VEL
LIN {X 0,Y 339.56,Z 388.926,A -85,B 0,C 180,E1 -14138.332,E2 -14138.332} C_VEL
LIN {X 0,Y 340.128,Z 382.557,A -85,B 0,C 180,E1 -14140.418,E2 -14140.418} C_VEL
LIN {X 0,Y 340.854,Z 375.626,A -85,B 0,C 180,E1 -14142.203,E2 -14142.203} C_VEL
LIN {X 0,Y 341.682,Z 368.556,A -85,B 0,C 180,E1 -14143.684,E2 -14143.684} C_VEL
LIN {X 0,Y 342.694,Z 360.045,A -85,B 0,C 180,E1 -14145.159,E2 -14145.159} C_VEL
LIN {X 0,Y 343.778,Z 349.516,A -85,B 0,C 180,E1 -14146.633,E2 -14146.633} C_VEL
LIN {X 0,Y 344.94,Z 339.116,A -85,B 0,C 180,E1 -14147.797,E2 -14147.797} C_VEL
LIN {X 0,Y 345.559,Z 331.26,A -85,B 0,C 180,E1 -14148.531,E2 -14148.531} C_VEL
LIN {X 0,Y 344.374,Z 319.44,A -85,B 0,C 180,E1 -14149.509,E2 -14149.509} C_VEL
LIN {X 0,Y 342.647,Z 305.922,A -85,B 0,C 180,E1 -14150.381,E2 -14150.381} C_VEL
LIN {X 0,Y 340.393,Z 292.915,A -85,B 0,C 180,E1 -14150.998,E2 -14150.998} C_VEL
LIN {X 0,Y 340.28,Z 291.748,A -85,B 0,C 180,E1 -14151.07,E2 -14151.07} C_VEL
LIN {X 0,Y 340.862,Z 284.221,A -85,B 0,C 180,E1 -14154.878,E2 -14154.878} C_VEL
LIN {X 0,Y 341.571,Z 277.594,A -85,B 0,C 180,E1 -14158.246,E2 -14158.246} C_VEL
LIN {X 0,Y 342.476,Z 269.921,A -85,B 0,C 180,E1 -14162.247,E2 -14162.247} C_VEL
LIN {X 0,Y 343.227,Z 263.468,A -85,B 0,C 180,E1 -14165.704,E2 -14165.704} C_VEL
LIN {X 0,Y 343.126,Z 259.583,A -85,B 0,C 180,E1 -14167.915,E2 -14167.915} C_VEL
LIN {X 0,Y 342.276,Z 254.423,A -85,B 0,C 180,E1 -14171.078,E2 -14171.078} C_VEL
LIN {X 0,Y 341.322,Z 249.272,A -85,B 0,C 180,E1 -14174.435,E2 -14174.435} C_VEL
LIN {X 0,Y 340.699,Z 246.05,A -85,B 0,C 180,E1 -14176.756,E2 -14176.756} C_VEL
LIN {X 0,Y 340.706,Z 246.047,A -85,B 0,C 180,E1 -14180.248,E2 -14180.248} C_VEL
LIN {X 0,Y 340.716,Z 246.041,A -85,B 0,C 180,E1 -14183.56,E2 -14183.56} C_VEL
LIN {X 0,Y 340.699,Z 246.046,A -85,B 0,C 180,E1 -14186.154,E2 -14186.154} C_VEL
LIN {X 0,Y 340.736,Z 246.043,A -85,B 0,C 180,E1 -14190.329,E2 -14190.329} C_VEL
LIN {X 0,Y 340.752,Z 246.042,A -85,B 0,C 180,E1 -14194.334,E2 -14194.334} C_VEL
LIN {X 0,Y 340.749,Z 246.042,A -85,B 0,C 180,E1 -14198.207,E2 -14198.207} C_VEL
LIN {X 0,Y 340.795,Z 246.036,A -85,B 0,C 180,E1 -14201.981,E2 -14201.981} C_VEL
LIN {X 0,Y 340.84,Z 246.029,A -85,B 0,C 180,E1 -14205.73,E2 -14205.73} C_VEL
LIN {X 0,Y 340.851,Z 246.026,A -85,B 0,C 180,E1 -14209.306,E2 -14209.306} C_VEL
LIN {X 0,Y 341.052,Z 245.999,A -85,B 0,C 180,E1 -14212.898,E2 -14212.898} C_VEL
LIN {X 0,Y 341.175,Z 245.989,A -85,B 0,C 180,E1 -14217.639,E2 -14217.639} C_VEL
LIN {X 0,Y 341.262,Z 245.974,A -85,B 0,C 180,E1 -14220,E2 -14220} C_VEL
LIN {X 0,Y 341.139,Z 245.988,A -85,B 0,C 180,E1 -14222.362,E2 -14222.362} C_VEL
LIN {X 0,Y 341.006,Z 246.008,A -85,B 0,C 180,E1 -14227.103,E2 -14227.103} C_VEL
LIN {X 0,Y 340.855,Z 246.025,A -85,B 0,C 180,E1 -14230.695,E2 -14230.695} C_VEL
LIN {X 0,Y 340.872,Z 246.021,A -85,B 0,C 180,E1 -14234.325,E2 -14234.325} C_VEL
LIN {X 0,Y 340.794,Z 246.032,A -85,B 0,C 180,E1 -14238.44,E2 -14238.44} C_VEL
LIN {X 0,Y 340.726,Z 246.04,A -85,B 0,C 180,E1 -14241.841,E2 -14241.841} C_VEL
LIN {X 0,Y 340.714,Z 246.047,A -85,B 0,C 180,E1 -14244.821,E2 -14244.821} C_VEL
LIN {X 0,Y 340.686,Z 246.047,A -85,B 0,C 180,E1 -14248.325,E2 -14248.325} C_VEL
LIN {X 0,Y 340.701,Z 246.045,A -85,B 0,C 180,E1 -14251.045,E2 -14251.045} C_VEL
LIN {X 0,Y 340.726,Z 246.04,A -85,B 0,C 180,E1 -14255.278,E2 -14255.278} C_VEL
LIN {X 0,Y 340.717,Z 246.047,A -85,B 0,C 180,E1 -14258.385,E2 -14258.385} C_VEL
LIN {X 0,Y 340.706,Z 246.046,A -85,B 0,C 180,E1 -14262.045,E2 -14262.045} C_VEL
LIN {X 0,Y 340.657,Z 246.053,A -85,B 0,C 180,E1 -14266.227,E2 -14266.227} C_VEL
LIN {X 0,Y 340.675,Z 246.047,A -85,B 0,C 180,E1 -14268.687,E2 -14268.687} C_VEL
LIN {X 0,Y 340.725,Z 246.044,A -85,B 0,C 180,E1 -14271.77,E2 -14271.77} C_VEL
LIN {X 0,Y 340.728,Z 246.043,A -85,B 0,C 180,E1 -14275.595,E2 -14275.595} C_VEL
LIN {X 0,Y 340.547,Z 246.061,A -85,B 0,C 180,E1 -14278.938,E2 -14278.938} C_VEL
LIN {X 0,Y 340.165,Z 246.115,A -85,B 0,C 180,E1 -14282.674,E2 -14282.674} C_VEL
LIN {X 0,Y 340.049,Z 248.558,A -85,B 0,C 180,E1 -14285.583,E2 -14285.583} C_VEL
LIN {X 0,Y 339.89,Z 252.022,A -85,B 0,C 180,E1 -14289.418,E2 -14289.418} C_VEL
LIN {X 0,Y 339.833,Z 255.713,A -85,B 0,C 180,E1 -14293.305,E2 -14293.305} C_VEL
LIN {X 0,Y 343.925,Z 270.656,A -85,B 0,C 180,E1 -14294.199,E2 -14294.199} C_VEL
LIN {X 0,Y 346.429,Z 281.949,A -85,B 0,C 180,E1 -14295.05,E2 -14295.05} C_VEL
LIN {X 0,Y 346.939,Z 285.072,A -85,B 0,C 180,E1 -14295.318,E2 -14295.318} C_VEL
LIN {X 0,Y 346.001,Z 297.136,A -85,B 0,C 180,E1 -14296.34,E2 -14296.34} C_VEL
LIN {X 0,Y 345.017,Z 307.742,A -85,B 0,C 180,E1 -14297.499,E2 -14297.499} C_VEL
LIN {X 0,Y 343.866,Z 318.108,A -85,B 0,C 180,E1 -14298.91,E2 -14298.91} C_VEL
LIN {X 0,Y 342.919,Z 326.206,A -85,B 0,C 180,E1 -14300.264,E2 -14300.264} C_VEL
LIN {X 0,Y 342.016,Z 334.783,A -85,B 0,C 180,E1 -14302.025,E2 -14302.025} C_VEL
LIN {X 0,Y 341.171,Z 341.637,A -85,B 0,C 180,E1 -14303.79,E2 -14303.79} C_VEL
LIN {X 0,Y 340.274,Z 347.937,A -85,B 0,C 180,E1 -14305.853,E2 -14305.853} C_VEL
LIN {X 0,Y 339.753,Z 352.076,A -85,B 0,C 180,E1 -14307.627,E2 -14307.627} C_VEL
LIN {X 0,Y 339.558,Z 354.271,A -85,B 0,C 180,E1 -14308.812,E2 -14308.812} C_VEL
LIN {X 0,Y 339.444,Z 355.991,A -85,B 0,C 180,E1 -14309.998,E2 -14309.998} C_VEL
LIN {X 0,Y 339.422,Z 357.297,A -85,B 0,C 180,E1 -14311.185,E2 -14311.185} C_VEL
LIN {X 0,Y 339.407,Z 358.222,A -85,B 0,C 180,E1 -14312.372,E2 -14312.372} C_VEL
LIN {X 0,Y 339.331,Z 358.77,A -85,B 0,C 180,E1 -14313.561,E2 -14313.561} C_VEL
LIN {X 0,Y 339.459,Z 358.621,A -85,B 0,C 180,E1 -14315.94,E2 -14315.94} C_VEL
LIN {X 0,Y 339.539,Z 357.977,A -85,B 0,C 180,E1 -14317.132,E2 -14317.132} C_VEL
LIN {X 0,Y 339.629,Z 356.95,A -85,B 0,C 180,E1 -14318.327,E2 -14318.327} C_VEL
LIN {X 0,Y 339.819,Z 355.472,A -85,B 0,C 180,E1 -14319.522,E2 -14319.522} C_VEL
LIN {X 0,Y 340.227,Z 352.474,A -85,B 0,C 180,E1 -14321.315,E2 -14321.315} C_VEL
LIN {X 0,Y 340.868,Z 348.417,A -85,B 0,C 180,E1 -14323.107,E2 -14323.107} C_VEL
LIN {X 0,Y 341.792,Z 342.379,A -85,B 0,C 180,E1 -14325.136,E2 -14325.136} C_VEL
LIN {X 0,Y 342.873,Z 335.363,A -85,B 0,C 180,E1 -14326.981,E2 -14326.981} C_VEL
LIN {X 0,Y 344.152,Z 326.801,A -85,B 0,C 180,E1 -14328.76,E2 -14328.76} C_VEL
LIN {X 0,Y 345.382,Z 317.984,A -85,B 0,C 180,E1 -14330.236,E2 -14330.236} C_VEL
LIN {X 0,Y 346.582,Z 308.27,A -85,B 0,C 180,E1 -14331.562,E2 -14331.562} C_VEL
LIN {X 0,Y 347.864,Z 297.617,A -85,B 0,C 180,E1 -14332.725,E2 -14332.725} C_VEL
LIN {X 0,Y 348.728,Z 287.258,A -85,B 0,C 180,E1 -14333.634,E2 -14333.634} C_VEL
LIN {X 0,Y 346.064,Z 275.718,A -85,B 0,C 180,E1 -14334.657,E2 -14334.657} C_VEL
LIN {X 0,Y 342.45,Z 263.497,A -85,B 0,C 180,E1 -14335.564,E2 -14335.564} C_VEL
LIN {X 0,Y 340.009,Z 256.044,A -85,B 0,C 180,E1 -14336.053,E2 -14336.053} C_VEL
LIN {X 0,Y 340.142,Z 252.676,A -85,B 0,C 180,E1 -14339.795,E2 -14339.795} C_VEL
LIN {X 0,Y 340.256,Z 250.368,A -85,B 0,C 180,E1 -14342.479,E2 -14342.479} C_VEL
LIN {X 0,Y 340.414,Z 247.118,A -85,B 0,C 180,E1 -14346.373,E2 -14346.373} C_VEL
LIN {X 0,Y 340.524,Z 246.069,A -85,B 0,C 180,E1 -14348.346,E2 -14348.346} C_VEL
LIN {X 0,Y 340.684,Z 246.048,A -85,B 0,C 180,E1 -14352.042,E2 -14352.042} C_VEL
LIN {X 0,Y 340.645,Z 246.056,A -85,B 0,C 180,E1 -14356.225,E2 -14356.225} C_VEL
LIN {X 0,Y 340.677,Z 246.049,A -85,B 0,C 180,E1 -14358.342,E2 -14358.342} C_VEL
LIN {X 0,Y 340.005,Z 246.134,A -85,B 0,C 180,E1 -14359.329,E2 -14359.329} C_VEL
LIN {X 0,Y 337.152,Z 246.488,A -85,B 0,C 180,E1 -14360.934,E2 -14360.934} C_VEL
LIN {X 0,Y 334.748,Z 246.788,A -85,B 0,C 180,E1 -14362.234,E2 -14362.234} C_VEL
LIN {X 0,Y 333.733,Z 246.911,A -85,B 0,C 180,E1 -14363.24,E2 -14363.24} C_VEL
LIN {X 0,Y 333.659,Z 246.92,A -85,B 0,C 180,E1 -14363.58,E2 -14363.58} C_VEL
LIN {X 0,Y 333.628,Z 246.925,A -85,B 0,C 180,E1 -14366.79,E2 -14366.79} C_VEL
LIN {X 0,Y 333.685,Z 246.919,A -85,B 0,C 180,E1 -14369.711,E2 -14369.711} C_VEL
LIN {X 0,Y 333.73,Z 246.911,A -85,B 0,C 180,E1 -14372.4,E2 -14372.4} C_VEL
LIN {X 0,Y 333.717,Z 246.915,A -85,B 0,C 180,E1 -14375.09,E2 -14375.09} C_VEL
LIN {X 0,Y 333.675,Z 246.923,A -85,B 0,C 180,E1 -14379.019,E2 -14379.019} C_VEL
LIN {X 0,Y 333.783,Z 246.906,A -85,B 0,C 180,E1 -14381.589,E2 -14381.589} C_VEL
LIN {X 0,Y 333.797,Z 246.908,A -85,B 0,C 180,E1 -14385.576,E2 -14385.576} C_VEL
LIN {X 0,Y 333.822,Z 246.904,A -85,B 0,C 180,E1 -14389.077,E2 -14389.077} C_VEL
LIN {X 0,Y 334.018,Z 246.877,A -85,B 0,C 180,E1 -14392.747,E2 -14392.747} C_VEL
LIN {X 0,Y 333.808,Z 246.906,A -85,B 0,C 180,E1 -14395.169,E2 -14395.169} C_VEL
LIN {X 0,Y 334.122,Z 246.865,A -85,B 0,C 180,E1 -14397.589,E2 -14397.589} C_VEL
LIN {X 0,Y 334.215,Z 246.854,A -85,B 0,C 180,E1 -14400,E2 -14400} C_VEL
LIN {X 0,Y 334.097,Z 246.869,A -85,B 0,C 180,E1 -14402.411,E2 -14402.411} C_VEL
LIN {X 0,Y 334.014,Z 246.878,A -85,B 0,C 180,E1 -14406.039,E2 -14406.039} C_VEL
LIN {X 0,Y 333.973,Z 246.885,A -85,B 0,C 180,E1 -14408.501,E2 -14408.501} C_VEL
LIN {X 0,Y 333.779,Z 246.908,A -85,B 0,C 180,E1 -14412.155,E2 -14412.155} C_VEL
LIN {X 0,Y 333.766,Z 246.905,A -85,B 0,C 180,E1 -14415.887,E2 -14415.887} C_VEL
LIN {X 0,Y 333.786,Z 246.904,A -85,B 0,C 180,E1 -14418.656,E2 -14418.656} C_VEL
LIN {X 0,Y 333.681,Z 246.921,A -85,B 0,C 180,E1 -14422.279,E2 -14422.279} C_VEL
LIN {X 0,Y 333.726,Z 246.914,A -85,B 0,C 180,E1 -14426.247,E2 -14426.247} C_VEL
LIN {X 0,Y 333.702,Z 246.919,A -85,B 0,C 180,E1 -14428.973,E2 -14428.973} C_VEL
LIN {X 0,Y 333.642,Z 246.925,A -85,B 0,C 180,E1 -14432.59,E2 -14432.59} C_VEL
LIN {X 0,Y 333.667,Z 246.923,A -85,B 0,C 180,E1 -14436.14,E2 -14436.14} C_VEL
LIN {X 0,Y 333.638,Z 246.924,A -85,B 0,C 180,E1 -14439.194,E2 -14439.194} C_VEL
LIN {X 0,Y 333.642,Z 246.974,A -85,B 0,C 180,E1 -14440.768,E2 -14440.768} C_VEL
LIN {X 0,Y 334.527,Z 251.664,A -85,B 0,C 180,E1 -14444.417,E2 -14444.417} C_VEL
LIN {X 0,Y 335.443,Z 256.549,A -85,B 0,C 180,E1 -14447.901,E2 -14447.901} C_VEL
LIN {X 0,Y 336.301,Z 261.467,A -85,B 0,C 180,E1 -14451.178,E2 -14451.178} C_VEL
LIN {X 0,Y 336.589,Z 265.179,A -85,B 0,C 180,E1 -14453.484,E2 -14453.484} C_VEL
LIN {X 0,Y 336.025,Z 270.053,A -85,B 0,C 180,E1 -14456.298,E2 -14456.298} C_VEL
LIN {X 0,Y 335.088,Z 276.297,A -85,B 0,C 180,E1 -14459.779,E2 -14459.779} C_VEL
LIN {X 0,Y 334.349,Z 282.485,A -85,B 0,C 180,E1 -14463.135,E2 -14463.135} C_VEL
LIN {X 0,Y 333.572,Z 289.873,A -85,B 0,C 180,E1 -14467.062,E2 -14467.062} C_VEL
LIN {X 0,Y 333.45,Z 291.153,A -85,B 0,C 180,E1 -14467.736,E2 -14467.736} C_VEL
LIN {X 0,Y 336.396,Z 305.064,A -85,B 0,C 180,E1 -14468.493,E2 -14468.493} C_VEL
LIN {X 0,Y 338.285,Z 317.954,A -85,B 0,C 180,E1 -14469.392,E2 -14469.392} C_VEL
LIN {X 0,Y 339.267,Z 330.123,A -85,B 0,C 180,E1 -14470.432,E2 -14470.432} C_VEL
LIN {X 0,Y 339.452,Z 335.577,A -85,B 0,C 180,E1 -14470.971,E2 -14470.971} C_VEL
LIN {X 0,Y 338.048,Z 346.5,A -85,B 0,C 180,E1 -14472.144,E2 -14472.144} C_VEL
LIN {X 0,Y 336.671,Z 356.684,A -85,B 0,C 180,E1 -14473.524,E2 -14473.524} C_VEL
LIN {X 0,Y 335.426,Z 366.288,A -85,B 0,C 180,E1 -14475.142,E2 -14475.142} C_VEL
LIN {X 0,Y 334.488,Z 373.548,A -85,B 0,C 180,E1 -14476.639,E2 -14476.639} C_VEL
LIN {X 0,Y 333.448,Z 380.773,A -85,B 0,C 180,E1 -14478.452,E2 -14478.452} C_VEL
LIN {X 0,Y 332.819,Z 386.564,A -85,B 0,C 180,E1 -14480.276,E2 -14480.276} C_VEL
LIN {X 0,Y 332.371,Z 391.139,A -85,B 0,C 180,E1 -14482.102,E2 -14482.102} C_VEL
LIN {X 0,Y 332.18,Z 394.634,A -85,B 0,C 180,E1 -14483.929,E2 -14483.929} C_VEL
LIN {X 0,Y 332.108,Z 396.384,A -85,B 0,C 180,E1 -14485.146,E2 -14485.146} C_VEL
LIN {X 0,Y 332.055,Z 397.722,A -85,B 0,C 180,E1 -14486.361,E2 -14486.361} C_VEL
LIN {X 0,Y 332.129,Z 399.211,A -85,B 0,C 180,E1 -14488.789,E2 -14488.789} C_VEL
LIN {X 0,Y 332.213,Z 399.319,A -85,B 0,C 180,E1 -14490.002,E2 -14490.002} C_VEL
LIN {X 0,Y 332.166,Z 399.026,A -85,B 0,C 180,E1 -14491.214,E2 -14491.214} C_VEL
LIN {X 0,Y 332.058,Z 397.252,A -85,B 0,C 180,E1 -14493.642,E2 -14493.642} C_VEL
LIN {X 0,Y 332.116,Z 395.709,A -85,B 0,C 180,E1 -14494.857,E2 -14494.857} C_VEL
LIN {X 0,Y 332.22,Z 392.593,A -85,B 0,C 180,E1 -14496.683,E2 -14496.683} C_VEL
LIN {X 0,Y 332.503,Z 388.408,A -85,B 0,C 180,E1 -14498.51,E2 -14498.51} C_VEL
LIN {X 0,Y 333.105,Z 382.016,A -85,B 0,C 180,E1 -14500.64,E2 -14500.64} C_VEL
LIN {X 0,Y 333.889,Z 375.06,A -85,B 0,C 180,E1 -14502.461,E2 -14502.461} C_VEL
LIN {X 0,Y 334.709,Z 367.958,A -85,B 0,C 180,E1 -14503.975,E2 -14503.975} C_VEL
LIN {X 0,Y 335.817,Z 359.057,A -85,B 0,C 180,E1 -14505.533,E2 -14505.533} C_VEL
LIN {X 0,Y 336.901,Z 348.817,A -85,B 0,C 180,E1 -14506.982,E2 -14506.982} C_VEL
LIN {X 0,Y 338.125,Z 338.362,A -85,B 0,C 180,E1 -14508.168,E2 -14508.168} C_VEL
LIN {X 0,Y 338.653,Z 332.156,A -85,B 0,C 180,E1 -14508.766,E2 -14508.766} C_VEL
LIN {X 0,Y 337.484,Z 319.864,A -85,B 0,C 180,E1 -14509.827,E2 -14509.827} C_VEL
LIN {X 0,Y 335.732,Z 306.047,A -85,B 0,C 180,E1 -14510.752,E2 -14510.752} C_VEL
LIN {X 0,Y 333.564,Z 293.47,A -85,B 0,C 180,E1 -14511.383,E2 -14511.383} C_VEL
LIN {X 0,Y 333.239,Z 291.371,A -85,B 0,C 180,E1 -14511.464,E2 -14511.464} C_VEL
LIN {X 0,Y 333.971,Z 283.396,A -85,B 0,C 180,E1 -14515.618,E2 -14515.618} C_VEL
LIN {X 0,Y 334.776,Z 275.885,A -85,B 0,C 180,E1 -14519.562,E2 -14519.562} C_VEL
LIN {X 0,Y 335.621,Z 269.286,A -85,B 0,C 180,E1 -14523.111,E2 -14523.111} C_VEL
LIN {X 0,Y 336.216,Z 264.361,A -85,B 0,C 180,E1 -14525.825,E2 -14525.825} C_VEL
LIN {X 0,Y 336.09,Z 260.492,A -85,B 0,C 180,E1 -14528.09,E2 -14528.09} C_VEL
LIN {X 0,Y 335.314,Z 255.788,A -85,B 0,C 180,E1 -14531.015,E2 -14531.015} C_VEL
LIN {X 0,Y 334.392,Z 250.732,A -85,B 0,C 180,E1 -14534.391,E2 -14534.391} C_VEL
LIN {X 0,Y 333.651,Z 246.929,A -85,B 0,C 180,E1 -14537.195,E2 -14537.195} C_VEL
LIN {X 0,Y 333.653,Z 246.926,A -85,B 0,C 180,E1 -14540.809,E2 -14540.809} C_VEL
LIN {X 0,Y 333.682,Z 246.918,A -85,B 0,C 180,E1 -14543.862,E2 -14543.862} C_VEL
LIN {X 0,Y 333.65,Z 246.921,A -85,B 0,C 180,E1 -14547.414,E2 -14547.414} C_VEL
LIN {X 0,Y 333.676,Z 246.919,A -85,B 0,C 180,E1 -14551.025,E2 -14551.025} C_VEL
LIN {X 0,Y 333.721,Z 246.912,A -85,B 0,C 180,E1 -14555.09,E2 -14555.09} C_VEL
LIN {X 0,Y 333.677,Z 246.918,A -85,B 0,C 180,E1 -14559.019,E2 -14559.019} C_VEL
LIN {X 0,Y 333.747,Z 246.911,A -85,B 0,C 180,E1 -14561.587,E2 -14561.587} C_VEL
LIN {X 0,Y 333.781,Z 246.907,A -85,B 0,C 180,E1 -14565.601,E2 -14565.601} C_VEL
LIN {X 0,Y 333.821,Z 246.9,A -85,B 0,C 180,E1 -14569.078,E2 -14569.078} C_VEL
LIN {X 0,Y 333.999,Z 246.877,A -85,B 0,C 180,E1 -14572.747,E2 -14572.747} C_VEL
LIN {X 0,Y 333.812,Z 246.903,A -85,B 0,C 180,E1 -14575.169,E2 -14575.169} C_VEL
LIN {X 0,Y 334.112,Z 246.869,A -85,B 0,C 180,E1 -14577.589,E2 -14577.589} C_VEL
LIN {X 0,Y 334.214,Z 246.852,A -85,B 0,C 180,E1 -14580,E2 -14580} C_VEL
LIN {X 0,Y 334.079,Z 246.868,A -85,B 0,C 180,E1 -14582.412,E2 -14582.412} C_VEL
LIN {X 0,Y 333.962,Z 246.882,A -85,B 0,C 180,E1 -14586.518,E2 -14586.518} C_VEL
LIN {X 0,Y 333.828,Z 246.9,A -85,B 0,C 180,E1 -14589.696,E2 -14589.696} C_VEL
LIN {X 0,Y 333.805,Z 246.905,A -85,B 0,C 180,E1 -14593.391,E2 -14593.391} C_VEL
LIN {X 0,Y 333.728,Z 246.916,A -85,B 0,C 180,E1 -14597.147,E2 -14597.147} C_VEL
LIN {X 0,Y 333.693,Z 246.915,A -85,B 0,C 180,E1 -14599.693,E2 -14599.693} C_VEL
LIN {X 0,Y 333.652,Z 246.921,A -85,B 0,C 180,E1 -14603.592,E2 -14603.592} C_VEL
LIN {X 0,Y 333.667,Z 246.919,A -85,B 0,C 180,E1 -14607.606,E2 -14607.606} C_VEL
LIN {X 0,Y 333.665,Z 246.922,A -85,B 0,C 180,E1 -14610.366,E2 -14610.366} C_VEL
LIN {X 0,Y 333.645,Z 246.922,A -85,B 0,C 180,E1 -14613.208,E2 -14613.208} C_VEL
LIN {X 0,Y 333.684,Z 246.92,A -85,B 0,C 180,E1 -14616.138,E2 -14616.138} C_VEL
LIN {X 0,Y 333.654,Z 246.921,A -85,B 0,C 180,E1 -14619.192,E2 -14619.192} C_VEL
LIN {X 0,Y 333.64,Z 246.926,A -85,B 0,C 180,E1 -14622.499,E2 -14622.499} C_VEL
LIN {X 0,Y 333.601,Z 246.931,A -85,B 0,C 180,E1 -14625.954,E2 -14625.954} C_VEL
LIN {X 0,Y 333.608,Z 246.927,A -85,B 0,C 180,E1 -14629.324,E2 -14629.324} C_VEL
LIN {X 0,Y 333.668,Z 246.919,A -85,B 0,C 180,E1 -14633.168,E2 -14633.168} C_VEL
LIN {X 0,Y 333.679,Z 246.919,A -85,B 0,C 180,E1 -14635.34,E2 -14635.34} C_VEL
LIN {X 0,Y 333.535,Z 246.937,A -85,B 0,C 180,E1 -14638.21,E2 -14638.21} C_VEL
LIN {X 0,Y 333.292,Z 246.965,A -85,B 0,C 180,E1 -14640.986,E2 -14640.986} C_VEL
LIN {X 0,Y 333.141,Z 246.989,A -85,B 0,C 180,E1 -14642.381,E2 -14642.381} C_VEL
LIN {X 0,Y 333.004,Z 249.105,A -85,B 0,C 180,E1 -14645.164,E2 -14645.164} C_VEL
LIN {X 0,Y 332.87,Z 252.467,A -85,B 0,C 180,E1 -14648.964,E2 -14648.964} C_VEL
LIN {X 0,Y 332.785,Z 256.124,A -85,B 0,C 180,E1 -14652.896,E2 -14652.896} C_VEL
LIN {X 0,Y 336.572,Z 269.767,A -85,B 0,C 180,E1 -14653.713,E2 -14653.713} C_VEL
LIN {X 0,Y 339.247,Z 281.144,A -85,B 0,C 180,E1 -14654.58,E2 -14654.58} C_VEL
LIN {X 0,Y 340.121,Z 286.037,A -85,B 0,C 180,E1 -14655.004,E2 -14655.004} C_VEL
LIN {X 0,Y 339.168,Z 298.084,A -85,B 0,C 180,E1 -14656.06,E2 -14656.06} C_VEL
LIN {X 0,Y 338.145,Z 308.581,A -85,B 0,C 180,E1 -14657.241,E2 -14657.241} C_VEL
LIN {X 0,Y 337.045,Z 318.174,A -85,B 0,C 180,E1 -14658.572,E2 -14658.572} C_VEL
LIN {X 0,Y 335.962,Z 326.939,A -85,B 0,C 180,E1 -14660.064,E2 -14660.064} C_VEL
LIN {X 0,Y 335.038,Z 335.432,A -85,B 0,C 180,E1 -14661.858,E2 -14661.858} C_VEL
LIN {X 0,Y 334.16,Z 342.24,A -85,B 0,C 180,E1 -14663.659,E2 -14663.659} C_VEL
LIN {X 0,Y 333.218,Z 348.506,A -85,B 0,C 180,E1 -14665.765,E2 -14665.765} C_VEL
LIN {X 0,Y 332.693,Z 352.612,A -85,B 0,C 180,E1 -14667.577,E2 -14667.577} C_VEL
LIN {X 0,Y 332.493,Z 354.785,A -85,B 0,C 180,E1 -14668.787,E2 -14668.787} C_VEL
LIN {X 0,Y 332.359,Z 357.772,A -85,B 0,C 180,E1 -14671.21,E2 -14671.21} C_VEL
LIN {X 0,Y 332.313,Z 358.685,A -85,B 0,C 180,E1 -14672.422,E2 -14672.422} C_VEL
LIN {X 0,Y 332.248,Z 359.211,A -85,B 0,C 180,E1 -14673.637,E2 -14673.637} C_VEL
LIN {X 0,Y 332.311,Z 359.308,A -85,B 0,C 180,E1 -14674.851,E2 -14674.851} C_VEL
LIN {X 0,Y 332.41,Z 358.889,A -85,B 0,C 180,E1 -14676.43,E2 -14676.43} C_VEL
LIN {X 0,Y 332.572,Z 357.321,A -85,B 0,C 180,E1 -14678.505,E2 -14678.505} C_VEL
LIN {X 0,Y 332.805,Z 355.82,A -85,B 0,C 180,E1 -14679.724,E2 -14679.724} C_VEL
LIN {X 0,Y 333.235,Z 352.792,A -85,B 0,C 180,E1 -14681.556,E2 -14681.556} C_VEL
LIN {X 0,Y 333.918,Z 348.702,A -85,B 0,C 180,E1 -14683.385,E2 -14683.385} C_VEL
LIN {X 0,Y 334.778,Z 343.329,A -85,B 0,C 180,E1 -14685.243,E2 -14685.243} C_VEL
LIN {X 0,Y 335.844,Z 336.798,A -85,B 0,C 180,E1 -14687.034,E2 -14687.034} C_VEL
LIN {X 0,Y 337.179,Z 328.54,A -85,B 0,C 180,E1 -14688.847,E2 -14688.847} C_VEL
LIN {X 0,Y 338.425,Z 320.014,A -85,B 0,C 180,E1 -14690.353,E2 -14690.353} C_VEL
LIN {X 0,Y 339.51,Z 311.427,A -85,B 0,C 180,E1 -14691.607,E2 -14691.607} C_VEL
LIN {X 0,Y 340.951,Z 300.378,A -85,B 0,C 180,E1 -14692.895,E2 -14692.895} C_VEL
LIN {X 0,Y 341.966,Z 290.259,A -85,B 0,C 180,E1 -14693.843,E2 -14693.843} C_VEL
LIN {X 0,Y 341.679,Z 286.957,A -85,B 0,C 180,E1 -14694.153,E2 -14694.153} C_VEL
LIN {X 0,Y 339.098,Z 275.983,A -85,B 0,C 180,E1 -14695.148,E2 -14695.148} C_VEL
LIN {X 0,Y 335.303,Z 263.549,A -85,B 0,C 180,E1 -14696.103,E2 -14696.103} C_VEL
LIN {X 0,Y 333.019,Z 256.497,A -85,B 0,C 180,E1 -14696.558,E2 -14696.558} C_VEL
LIN {X 0,Y 333.104,Z 253.093,A -85,B 0,C 180,E1 -14700.42,E2 -14700.42} C_VEL
LIN {X 0,Y 333.259,Z 250.743,A -85,B 0,C 180,E1 -14703.249,E2 -14703.249} C_VEL
LIN {X 0,Y 333.414,Z 247.82,A -85,B 0,C 180,E1 -14706.774,E2 -14706.774} C_VEL
LIN {X 0,Y 333.407,Z 247.107,A -85,B 0,C 180,E1 -14707.681,E2 -14707.681} C_VEL
LIN {X 0,Y 333.585,Z 246.932,A -85,B 0,C 180,E1 -14710.774,E2 -14710.774} C_VEL
LIN {X 0,Y 333.586,Z 246.934,A -85,B 0,C 180,E1 -14714.249,E2 -14714.249} C_VEL
LIN {X 0,Y 333.634,Z 246.928,A -85,B 0,C 180,E1 -14717.617,E2 -14717.617} C_VEL
LIN {X 0,Y 333.646,Z 246.925,A -85,B 0,C 180,E1 -14721.2,E2 -14721.2} C_VEL
LIN {X 0,Y 333.659,Z 246.92,A -85,B 0,C 180,E1 -14723.58,E2 -14723.58} C_VEL
LIN {X 0,Y 332.997,Z 247.007,A -85,B 0,C 180,E1 -14724.589,E2 -14724.589} C_VEL
LIN {X 0,Y 330.095,Z 247.369,A -85,B 0,C 180,E1 -14726.228,E2 -14726.228} C_VEL
LIN {X 0,Y 327.653,Z 247.674,A -85,B 0,C 180,E1 -14727.556,E2 -14727.556} C_VEL
LIN {X 0,Y 326.643,Z 247.796,A -85,B 0,C 180,E1 -14728.586,E2 -14728.586} C_VEL
LIN {X 0,Y 326.582,Z 247.803,A -85,B 0,C 180,E1 -14728.934,E2 -14728.934} C_VEL
LIN {X 0,Y 326.647,Z 247.795,A -85,B 0,C 180,E1 -14731.897,E2 -14731.897} C_VEL
LIN {X 0,Y 326.678,Z 247.793,A -85,B 0,C 180,E1 -14734.626,E2 -14734.626} C_VEL
LIN {X 0,Y 326.638,Z 247.798,A -85,B 0,C 180,E1 -14738.544,E2 -14738.544} C_VEL
LIN {X 0,Y 326.734,Z 247.785,A -85,B 0,C 180,E1 -14741.177,E2 -14741.177} C_VEL
LIN {X 0,Y 326.752,Z 247.785,A -85,B 0,C 180,E1 -14745.432,E2 -14745.432} C_VEL
LIN {X 0,Y 326.758,Z 247.783,A -85,B 0,C 180,E1 -14748.838,E2 -14748.838} C_VEL
LIN {X 0,Y 326.968,Z 247.756,A -85,B 0,C 180,E1 -14752.59,E2 -14752.59} C_VEL
LIN {X 0,Y 326.774,Z 247.781,A -85,B 0,C 180,E1 -14755.065,E2 -14755.065} C_VEL
LIN {X 0,Y 327.059,Z 247.745,A -85,B 0,C 180,E1 -14757.537,E2 -14757.537} C_VEL
LIN {X 0,Y 327.167,Z 247.732,A -85,B 0,C 180,E1 -14760,E2 -14760} C_VEL
LIN {X 0,Y 327.037,Z 247.749,A -85,B 0,C 180,E1 -14762.463,E2 -14762.463} C_VEL
LIN {X 0,Y 326.989,Z 247.753,A -85,B 0,C 180,E1 -14766.169,E2 -14766.169} C_VEL
LIN {X 0,Y 326.903,Z 247.765,A -85,B 0,C 180,E1 -14768.655,E2 -14768.655} C_VEL
LIN {X 0,Y 326.723,Z 247.785,A -85,B 0,C 180,E1 -14772.422,E2 -14772.422} C_VEL
LIN {X 0,Y 326.743,Z 247.781,A -85,B 0,C 180,E1 -14774.958,E2 -14774.958} C_VEL
LIN {X 0,Y 326.722,Z 247.783,A -85,B 0,C 180,E1 -14778.839,E2 -14778.839} C_VEL
LIN {X 0,Y 326.61,Z 247.801,A -85,B 0,C 180,E1 -14782.788,E2 -14782.788} C_VEL
LIN {X 0,Y 326.68,Z 247.793,A -85,B 0,C 180,E1 -14785.485,E2 -14785.485} C_VEL
LIN {X 0,Y 326.652,Z 247.797,A -85,B 0,C 180,E1 -14789.66,E2 -14789.66} C_VEL
LIN {X 0,Y 326.613,Z 247.802,A -85,B 0,C 180,E1 -14792.949,E2 -14792.949} C_VEL
LIN {X 0,Y 326.603,Z 247.799,A -85,B 0,C 180,E1 -14795.521,E2 -14795.521} C_VEL
LIN {X 0,Y 326.602,Z 247.801,A -85,B 0,C 180,E1 -14799.229,E2 -14799.229} C_VEL
LIN {X 0,Y 326.605,Z 247.907,A -85,B 0,C 180,E1 -14800.207,E2 -14800.207} C_VEL
LIN {X 0,Y 327.552,Z 252.854,A -85,B 0,C 180,E1 -14804.167,E2 -14804.167} C_VEL
LIN {X 0,Y 328.409,Z 257.501,A -85,B 0,C 180,E1 -14807.586,E2 -14807.586} C_VEL
LIN {X 0,Y 329.314,Z 262.529,A -85,B 0,C 180,E1 -14811.024,E2 -14811.024} C_VEL
LIN {X 0,Y 329.6,Z 266.165,A -85,B 0,C 180,E1 -14813.344,E2 -14813.344} C_VEL
LIN {X 0,Y 328.938,Z 271.392,A -85,B 0,C 180,E1 -14816.436,E2 -14816.436} C_VEL
LIN {X 0,Y 328.034,Z 277.245,A -85,B 0,C 180,E1 -14819.772,E2 -14819.772} C_VEL
LIN {X 0,Y 327.257,Z 283.4,A -85,B 0,C 180,E1 -14823.195,E2 -14823.195} C_VEL
LIN {X 0,Y 326.47,Z 290.901,A -85,B 0,C 180,E1 -14827.204,E2 -14827.204} C_VEL
LIN {X 0,Y 329.451,Z 304.52,A -85,B 0,C 180,E1 -14827.97,E2 -14827.97} C_VEL
LIN {X 0,Y 331.43,Z 317.586,A -85,B 0,C 180,E1 -14828.911,E2 -14828.911} C_VEL
LIN {X 0,Y 332.436,Z 330.238,A -85,B 0,C 180,E1 -14830.025,E2 -14830.025} C_VEL
LIN {X 0,Y 332.556,Z 336.994,A -85,B 0,C 180,E1 -14830.721,E2 -14830.721} C_VEL
LIN {X 0,Y 330.922,Z 348.694,A -85,B 0,C 180,E1 -14832.067,E2 -14832.067} C_VEL
LIN {X 0,Y 329.695,Z 357.556,A -85,B 0,C 180,E1 -14833.341,E2 -14833.341} C_VEL
LIN {X 0,Y 328.521,Z 366.198,A -85,B 0,C 180,E1 -14834.852,E2 -14834.852} C_VEL
LIN {X 0,Y 327.34,Z 374.586,A -85,B 0,C 180,E1 -14836.658,E2 -14836.658} C_VEL
LIN {X 0,Y 326.318,Z 381.49,A -85,B 0,C 180,E1 -14838.511,E2 -14838.511} C_VEL
LIN {X 0,Y 325.608,Z 387.86,A -85,B 0,C 180,E1 -14840.686,E2 -14840.686} C_VEL
LIN {X 0,Y 325.203,Z 392.041,A -85,B 0,C 180,E1 -14842.552,E2 -14842.552} C_VEL
LIN {X 0,Y 325.081,Z 394.529,A -85,B 0,C 180,E1 -14843.981,E2 -14843.981} C_VEL
LIN {X 0,Y 324.983,Z 397.326,A -85,B 0,C 180,E1 -14846.282,E2 -14846.282} C_VEL
LIN {X 0,Y 324.939,Z 398.259,A -85,B 0,C 180,E1 -14847.523,E2 -14847.523} C_VEL
LIN {X 0,Y 325.035,Z 398.79,A -85,B 0,C 180,E1 -14848.763,E2 -14848.763} C_VEL
LIN {X 0,Y 325.137,Z 398.888,A -85,B 0,C 180,E1 -14850.002,E2 -14850.002} C_VEL
LIN {X 0,Y 325.072,Z 398.585,A -85,B 0,C 180,E1 -14851.241,E2 -14851.241} C_VEL
LIN {X 0,Y 324.987,Z 396.789,A -85,B 0,C 180,E1 -14853.722,E2 -14853.722} C_VEL
LIN {X 0,Y 325.084,Z 393.568,A -85,B 0,C 180,E1 -14856.024,E2 -14856.024} C_VEL
LIN {X 0,Y 325.329,Z 389.407,A -85,B 0,C 180,E1 -14858.074,E2 -14858.074} C_VEL
LIN {X 0,Y 325.802,Z 384.433,A -85,B 0,C 180,E1 -14859.939,E2 -14859.939} C_VEL
LIN {X 0,Y 326.436,Z 378.167,A -85,B 0,C 180,E1 -14861.804,E2 -14861.804} C_VEL
LIN {X 0,Y 327.45,Z 370.371,A -85,B 0,C 180,E1 -14863.658,E2 -14863.658} C_VEL
LIN {X 0,Y 328.589,Z 361.327,A -85,B 0,C 180,E1 -14865.378,E2 -14865.378} C_VEL
LIN {X 0,Y 329.701,Z 351.562,A -85,B 0,C 180,E1 -14866.886,E2 -14866.886} C_VEL
LIN {X 0,Y 330.865,Z 341.838,A -85,B 0,C 180,E1 -14868.1,E2 -14868.1} C_VEL
LIN {X 0,Y 331.742,Z 332.956,A -85,B 0,C 180,E1 -14869.011,E2 -14869.011} C_VEL
LIN {X 0,Y 330.58,Z 320.408,A -85,B 0,C 180,E1 -14870.151,E2 -14870.151} C_VEL
LIN {X 0,Y 328.973,Z 307.145,A -85,B 0,C 180,E1 -14871.079,E2 -14871.079} C_VEL
LIN {X 0,Y 326.73,Z 293.875,A -85,B 0,C 180,E1 -14871.784,E2 -14871.784} C_VEL
LIN {X 0,Y 326.221,Z 290.921,A -85,B 0,C 180,E1 -14871.927,E2 -14871.927} C_VEL
LIN {X 0,Y 327.007,Z 283.044,A -85,B 0,C 180,E1 -14876.143,E2 -14876.143} C_VEL
LIN {X 0,Y 327.874,Z 275.444,A -85,B 0,C 180,E1 -14880.248,E2 -14880.248} C_VEL
LIN {X 0,Y 328.704,Z 269.09,A -85,B 0,C 180,E1 -14883.775,E2 -14883.775} C_VEL
LIN {X 0,Y 329.178,Z 265.559,A -85,B 0,C 180,E1 -14885.776,E2 -14885.776} C_VEL
LIN {X 0,Y 329.062,Z 261.377,A -85,B 0,C 180,E1 -14888.272,E2 -14888.272} C_VEL
LIN {X 0,Y 328.161,Z 256.201,A -85,B 0,C 180,E1 -14891.6,E2 -14891.6} C_VEL
LIN {X 0,Y 327.204,Z 251.061,A -85,B 0,C 180,E1 -14895.14,E2 -14895.14} C_VEL
LIN {X 0,Y 326.615,Z 247.805,A -85,B 0,C 180,E1 -14897.576,E2 -14897.576} C_VEL
LIN {X 0,Y 326.604,Z 247.801,A -85,B 0,C 180,E1 -14901.389,E2 -14901.389} C_VEL
LIN {X 0,Y 326.626,Z 247.8,A -85,B 0,C 180,E1 -14904.852,E2 -14904.852} C_VEL
LIN {X 0,Y 326.615,Z 247.798,A -85,B 0,C 180,E1 -14907.456,E2 -14907.456} C_VEL
LIN {X 0,Y 326.631,Z 247.801,A -85,B 0,C 180,E1 -14910.338,E2 -14910.338} C_VEL
LIN {X 0,Y 326.636,Z 247.795,A -85,B 0,C 180,E1 -14913.138,E2 -14913.138} C_VEL
LIN {X 0,Y 326.652,Z 247.795,A -85,B 0,C 180,E1 -14915.871,E2 -14915.871} C_VEL
LIN {X 0,Y 326.629,Z 247.799,A -85,B 0,C 180,E1 -14919.863,E2 -14919.863} C_VEL
LIN {X 0,Y 326.688,Z 247.792,A -85,B 0,C 180,E1 -14923.76,E2 -14923.76} C_VEL
LIN {X 0,Y 326.75,Z 247.783,A -85,B 0,C 180,E1 -14926.314,E2 -14926.314} C_VEL
LIN {X 0,Y 326.789,Z 247.779,A -85,B 0,C 180,E1 -14930.093,E2 -14930.093} C_VEL
LIN {X 0,Y 326.989,Z 247.756,A -85,B 0,C 180,E1 -14933.831,E2 -14933.831} C_VEL
LIN {X 0,Y 327.053,Z 247.748,A -85,B 0,C 180,E1 -14937.537,E2 -14937.537} C_VEL
LIN {X 0,Y 327.166,Z 247.73,A -85,B 0,C 180,E1 -14940,E2 -14940} C_VEL
LIN {X 0,Y 327.023,Z 247.747,A -85,B 0,C 180,E1 -14942.464,E2 -14942.464} C_VEL
LIN {X 0,Y 326.924,Z 247.758,A -85,B 0,C 180,E1 -14946.507,E2 -14946.507} C_VEL
LIN {X 0,Y 326.79,Z 247.775,A -85,B 0,C 180,E1 -14949.907,E2 -14949.907} C_VEL
LIN {X 0,Y 326.767,Z 247.779,A -85,B 0,C 180,E1 -14953.685,E2 -14953.685} C_VEL
LIN {X 0,Y 326.672,Z 247.792,A -85,B 0,C 180,E1 -14957.53,E2 -14957.53} C_VEL
LIN {X 0,Y 326.637,Z 247.794,A -85,B 0,C 180,E1 -14960.137,E2 -14960.137} C_VEL
LIN {X 0,Y 326.6,Z 247.805,A -85,B 0,C 180,E1 -14962.789,E2 -14962.789} C_VEL
LIN {X 0,Y 326.604,Z 247.803,A -85,B 0,C 180,E1 -14966.865,E2 -14966.865} C_VEL
LIN {X 0,Y 326.619,Z 247.802,A -85,B 0,C 180,E1 -14970.602,E2 -14970.602} C_VEL
LIN {X 0,Y 326.615,Z 247.798,A -85,B 0,C 180,E1 -14974.019,E2 -14974.019} C_VEL
LIN {X 0,Y 326.635,Z 247.795,A -85,B 0,C 180,E1 -14977.238,E2 -14977.238} C_VEL
LIN {X 0,Y 326.585,Z 247.802,A -85,B 0,C 180,E1 -14981.13,E2 -14981.13} C_VEL
LIN {X 0,Y 326.533,Z 247.809,A -85,B 0,C 180,E1 -14984.742,E2 -14984.742} C_VEL
LIN {X 0,Y 326.567,Z 247.809,A -85,B 0,C 180,E1 -14988.151,E2 -14988.151} C_VEL
LIN {X 0,Y 326.574,Z 247.804,A -85,B 0,C 180,E1 -14991.382,E2 -14991.382} C_VEL
LIN {X 0,Y 326.624,Z 247.797,A -85,B 0,C 180,E1 -14994.851,E2 -14994.851} C_VEL
LIN {X 0,Y 326.568,Z 247.805,A -85,B 0,C 180,E1 -14997.449,E2 -14997.449} C_VEL
LIN {X 0,Y 326.29,Z 247.838,A -85,B 0,C 180,E1 -15000.302,E2 -15000.302} C_VEL
LIN {X 0,Y 326.13,Z 247.862,A -85,B 0,C 180,E1 -15002.073,E2 -15002.073} C_VEL
LIN {X 0,Y 326.023,Z 248.273,A -85,B 0,C 180,E1 -15003.082,E2 -15003.082} C_VEL
LIN {X 0,Y 325.911,Z 250.576,A -85,B 0,C 180,E1 -15005.811,E2 -15005.811} C_VEL
LIN {X 0,Y 325.866,Z 252.912,A -85,B 0,C 180,E1 -15008.49,E2 -15008.49} C_VEL
LIN {X 0,Y 325.748,Z 256.556,A -85,B 0,C 180,E1 -15012.445,E2 -15012.445} C_VEL
LIN {X 0,Y 329.85,Z 271.126,A -85,B 0,C 180,E1 -15013.365,E2 -15013.365} C_VEL
LIN {X 0,Y 332.396,Z 282.131,A -85,B 0,C 180,E1 -15014.237,E2 -15014.237} C_VEL
LIN {X 0,Y 333.297,Z 287.032,A -85,B 0,C 180,E1 -15014.679,E2 -15014.679} C_VEL
LIN {X 0,Y 332.328,Z 299.012,A -85,B 0,C 180,E1 -15015.767,E2 -15015.767} C_VEL
LIN {X 0,Y 331.289,Z 309.417,A -85,B 0,C 180,E1 -15016.972,E2 -15016.972} C_VEL
LIN {X 0,Y 330.136,Z 318.95,A -85,B 0,C 180,E1 -15018.331,E2 -15018.331} C_VEL
LIN {X 0,Y 329.01,Z 327.669,A -85,B 0,C 180,E1 -15019.855,E2 -15019.855} C_VEL
LIN {X 0,Y 328.059,Z 336.073,A -85,B 0,C 180,E1 -15021.684,E2 -15021.684} C_VEL
LIN {X 0,Y 327.197,Z 341.847,A -85,B 0,C 180,E1 -15023.214,E2 -15023.214} C_VEL
LIN {X 0,Y 326.363,Z 347.482,A -85,B 0,C 180,E1 -15025.057,E2 -15025.057} C_VEL
LIN {X 0,Y 325.823,Z 351.916,A -85,B 0,C 180,E1 -15026.907,E2 -15026.907} C_VEL
LIN {X 0,Y 325.429,Z 355.294,A -85,B 0,C 180,E1 -15028.761,E2 -15028.761} C_VEL
LIN {X 0,Y 325.298,Z 358.247,A -85,B 0,C 180,E1 -15031.236,E2 -15031.236} C_VEL
LIN {X 0,Y 325.22,Z 359.148,A -85,B 0,C 180,E1 -15032.475,E2 -15032.475} C_VEL
LIN {X 0,Y 325.169,Z 359.647,A -85,B 0,C 180,E1 -15033.716,E2 -15033.716} C_VEL
LIN {X 0,Y 325.251,Z 359.727,A -85,B 0,C 180,E1 -15034.956,E2 -15034.956} C_VEL
LIN {X 0,Y 325.413,Z 358.763,A -85,B 0,C 180,E1 -15037.444,E2 -15037.444} C_VEL
LIN {X 0,Y 325.538,Z 357.688,A -85,B 0,C 180,E1 -15038.69,E2 -15038.69} C_VEL
LIN {X 0,Y 325.768,Z 356.17,A -85,B 0,C 180,E1 -15039.936,E2 -15039.936} C_VEL
LIN {X 0,Y 326.227,Z 353.112,A -85,B 0,C 180,E1 -15041.808,E2 -15041.808} C_VEL
LIN {X 0,Y 326.975,Z 348.988,A -85,B 0,C 180,E1 -15043.674,E2 -15043.674} C_VEL
LIN {X 0,Y 328.026,Z 342.779,A -85,B 0,C 180,E1 -15045.819,E2 -15045.819} C_VEL
LIN {X 0,Y 329.236,Z 335.774,A -85,B 0,C 180,E1 -15047.707,E2 -15047.707} C_VEL
LIN {X 0,Y 330.649,Z 327.079,A -85,B 0,C 180,E1 -15049.556,E2 -15049.556} C_VEL
LIN {X 0,Y 331.957,Z 318.147,A -85,B 0,C 180,E1 -15051.093,E2 -15051.093} C_VEL
LIN {X 0,Y 333.355,Z 308.291,A -85,B 0,C 180,E1 -15052.463,E2 -15052.463} C_VEL
LIN {X 0,Y 334.719,Z 297.654,A -85,B 0,C 180,E1 -15053.641,E2 -15053.641} C_VEL
LIN {X 0,Y 335.342,Z 291.044,A -85,B 0,C 180,E1 -15054.253,E2 -15054.253} C_VEL
LIN {X 0,Y 333.731,Z 282.432,A -85,B 0,C 180,E1 -15055.104,E2 -15055.104} C_VEL
LIN {X 0,Y 330.375,Z 270.223,A -85,B 0,C 180,E1 -15056.162,E2 -15056.162} C_VEL
LIN {X 0,Y 325.969,Z 256.914,A -85,B 0,C 180,E1 -15057.14,E2 -15057.14} C_VEL
LIN {X 0,Y 326.105,Z 253.46,A -85,B 0,C 180,E1 -15061.144,E2 -15061.144} C_VEL
LIN {X 0,Y 326.253,Z 251.058,A -85,B 0,C 180,E1 -15064.059,E2 -15064.059} C_VEL
LIN {X 0,Y 326.389,Z 248.551,A -85,B 0,C 180,E1 -15067.183,E2 -15067.183} C_VEL
LIN {X 0,Y 326.487,Z 247.816,A -85,B 0,C 180,E1 -15069.2,E2 -15069.2} C_VEL
LIN {X 0,Y 326.566,Z 247.809,A -85,B 0,C 180,E1 -15072.969,E2 -15072.969} C_VEL
LIN {X 0,Y 326.568,Z 247.807,A -85,B 0,C 180,E1 -15077.026,E2 -15077.026} C_VEL
LIN {X 0,Y 326.604,Z 247.802,A -85,B 0,C 180,E1 -15080.771,E2 -15080.771} C_VEL
LIN {X 0,Y 326.605,Z 247.804,A -85,B 0,C 180,E1 -15084.479,E2 -15084.479} C_VEL
LIN {X 0,Y 326.598,Z 247.804,A -85,B 0,C 180,E1 -15087.454,E2 -15087.454} C_VEL
LIN {X 0,Y 326.582,Z 247.803,A -85,B 0,C 180,E1 -15088.934,E2 -15088.934} C_VEL
LIN {X 0,Y 325.988,Z 247.877,A -85,B 0,C 180,E1 -15089.964,E2 -15089.964} C_VEL
LIN {X 0,Y 323.211,Z 248.228,A -85,B 0,C 180,E1 -15091.642,E2 -15091.642} C_VEL
LIN {X 0,Y 320.797,Z 248.531,A -85,B 0,C 180,E1 -15093.001,E2 -15093.001} C_VEL
LIN {X 0,Y 319.725,Z 248.662,A -85,B 0,C 180,E1 -15094.053,E2 -15094.053} C_VEL
LIN {X 0,Y 319.621,Z 248.673,A -85,B 0,C 180,E1 -15094.409,E2 -15094.409} C_VEL
LIN {X 0,Y 319.587,Z 248.676,A -85,B 0,C 180,E1 -15098.047,E2 -15098.047} C_VEL
LIN {X 0,Y 319.678,Z 248.665,A -85,B 0,C 180,E1 -15100.961,E2 -15100.961} C_VEL
LIN {X 0,Y 319.72,Z 248.66,A -85,B 0,C 180,E1 -15105.275,E2 -15105.275} C_VEL
LIN {X 0,Y 319.746,Z 248.656,A -85,B 0,C 180,E1 -15109.872,E2 -15109.872} C_VEL
LIN {X 0,Y 319.925,Z 248.635,A -85,B 0,C 180,E1 -15112.426,E2 -15112.426} C_VEL
LIN {X 0,Y 319.743,Z 248.657,A -85,B 0,C 180,E1 -15114.956,E2 -15114.956} C_VEL
LIN {X 0,Y 319.999,Z 248.625,A -85,B 0,C 180,E1 -15117.482,E2 -15117.482} C_VEL
LIN {X 0,Y 320.119,Z 248.61,A -85,B 0,C 180,E1 -15120,E2 -15120} C_VEL
LIN {X 0,Y 319.981,Z 248.627,A -85,B 0,C 180,E1 -15122.518,E2 -15122.518} C_VEL
LIN {X 0,Y 319.944,Z 248.631,A -85,B 0,C 180,E1 -15126.305,E2 -15126.305} C_VEL
LIN {X 0,Y 319.831,Z 248.646,A -85,B 0,C 180,E1 -15128.848,E2 -15128.848} C_VEL
LIN {X 0,Y 319.67,Z 248.663,A -85,B 0,C 180,E1 -15132.7,E2 -15132.7} C_VEL
LIN {X 0,Y 319.688,Z 248.658,A -85,B 0,C 180,E1 -15135.296,E2 -15135.296} C_VEL
LIN {X 0,Y 319.664,Z 248.662,A -85,B 0,C 180,E1 -15139.256,E2 -15139.256} C_VEL
LIN {X 0,Y 319.56,Z 248.68,A -85,B 0,C 180,E1 -15143.32,E2 -15143.32} C_VEL
LIN {X 0,Y 319.625,Z 248.671,A -85,B 0,C 180,E1 -15146.089,E2 -15146.089} C_VEL
LIN {X 0,Y 319.588,Z 248.677,A -85,B 0,C 180,E1 -15148.934,E2 -15148.934} C_VEL
LIN {X 0,Y 319.529,Z 248.685,A -85,B 0,C 180,E1 -15151.862,E2 -15151.862} C_VEL
LIN {X 0,Y 319.57,Z 248.675,A -85,B 0,C 180,E1 -15155.544,E2 -15155.544} C_VEL
LIN {X 0,Y 319.573,Z 248.833,A -85,B 0,C 180,E1 -15159.625,E2 -15159.625} C_VEL
LIN {X 0,Y 320.458,Z 253.681,A -85,B 0,C 180,E1 -15163.64,E2 -15163.64} C_VEL
LIN {X 0,Y 321.375,Z 258.533,A -85,B 0,C 180,E1 -15167.321,E2 -15167.321} C_VEL
LIN {X 0,Y 322.265,Z 263.444,A -85,B 0,C 180,E1 -15170.773,E2 -15170.773} C_VEL
LIN {X 0,Y 322.596,Z 267.064,A -85,B 0,C 180,E1 -15173.143,E2 -15173.143} C_VEL
LIN {X 0,Y 322.017,Z 271.799,A -85,B 0,C 180,E1 -15176.032,E2 -15176.032} C_VEL
LIN {X 0,Y 320.999,Z 278.176,A -85,B 0,C 180,E1 -15179.766,E2 -15179.766} C_VEL
LIN {X 0,Y 320.175,Z 284.301,A -85,B 0,C 180,E1 -15183.26,E2 -15183.26} C_VEL
LIN {X 0,Y 319.482,Z 290.289,A -85,B 0,C 180,E1 -15186.622,E2 -15186.622} C_VEL
LIN {X 0,Y 322.509,Z 304.038,A -85,B 0,C 180,E1 -15187.425,E2 -15187.425} C_VEL
LIN {X 0,Y 324.451,Z 316.034,A -85,B 0,C 180,E1 -15188.312,E2 -15188.312} C_VEL
LIN {X 0,Y 325.479,Z 328.249,A -85,B 0,C 180,E1 -15189.394,E2 -15189.394} C_VEL
LIN {X 0,Y 325.831,Z 336.9,A -85,B 0,C 180,E1 -15190.307,E2 -15190.307} C_VEL
LIN {X 0,Y 324.184,Z 348.541,A -85,B 0,C 180,E1 -15191.681,E2 -15191.681} C_VEL
LIN {X 0,Y 322.636,Z 358.881,A -85,B 0,C 180,E1 -15193.226,E2 -15193.226} C_VEL
LIN {X 0,Y 321.432,Z 367.294,A -85,B 0,C 180,E1 -15194.791,E2 -15194.791} C_VEL
LIN {X 0,Y 320.204,Z 375.539,A -85,B 0,C 180,E1 -15196.678,E2 -15196.678} C_VEL
LIN {X 0,Y 319.184,Z 382.194,A -85,B 0,C 180,E1 -15198.572,E2 -15198.572} C_VEL
LIN {X 0,Y 318.57,Z 387.523,A -85,B 0,C 180,E1 -15200.478,E2 -15200.478} C_VEL
LIN {X 0,Y 318.138,Z 391.682,A -85,B 0,C 180,E1 -15202.385,E2 -15202.385} C_VEL
LIN {X 0,Y 318.004,Z 394.369,A -85,B 0,C 180,E1 -15203.998,E2 -15203.998} C_VEL
LIN {X 0,Y 317.912,Z 396.931,A -85,B 0,C 180,E1 -15206.199,E2 -15206.199} C_VEL
LIN {X 0,Y 317.855,Z 397.855,A -85,B 0,C 180,E1 -15207.467,E2 -15207.467} C_VEL
LIN {X 0,Y 317.941,Z 398.367,A -85,B 0,C 180,E1 -15208.735,E2 -15208.735} C_VEL
LIN {X 0,Y 318.048,Z 398.456,A -85,B 0,C 180,E1 -15210.002,E2 -15210.002} C_VEL
LIN {X 0,Y 317.978,Z 398.144,A -85,B 0,C 180,E1 -15211.268,E2 -15211.268} C_VEL
LIN {X 0,Y 317.88,Z 397.438,A -85,B 0,C 180,E1 -15212.536,E2 -15212.536} C_VEL
LIN {X 0,Y 317.918,Z 396.323,A -85,B 0,C 180,E1 -15213.804,E2 -15213.804} C_VEL
LIN {X 0,Y 318.006,Z 393.34,A -85,B 0,C 180,E1 -15216.006,E2 -15216.006} C_VEL
LIN {X 0,Y 318.265,Z 388.896,A -85,B 0,C 180,E1 -15218.254,E2 -15218.254} C_VEL
LIN {X 0,Y 318.754,Z 383.897,A -85,B 0,C 180,E1 -15220.161,E2 -15220.161} C_VEL
LIN {X 0,Y 319.455,Z 377.609,A -85,B 0,C 180,E1 -15222.066,E2 -15222.066} C_VEL
LIN {X 0,Y 320.482,Z 369.766,A -85,B 0,C 180,E1 -15223.961,E2 -15223.961} C_VEL
LIN {X 0,Y 321.65,Z 361.091,A -85,B 0,C 180,E1 -15225.646,E2 -15225.646} C_VEL
LIN {X 0,Y 322.838,Z 350.879,A -85,B 0,C 180,E1 -15227.256,E2 -15227.256} C_VEL
LIN {X 0,Y 324.244,Z 339.712,A -85,B 0,C 180,E1 -15228.647,E2 -15228.647} C_VEL
LIN {X 0,Y 324.82,Z 333.747,A -85,B 0,C 180,E1 -15229.268,E2 -15229.268} C_VEL
LIN {X 0,Y 323.707,Z 321.175,A -85,B 0,C 180,E1 -15230.464,E2 -15230.464} C_VEL
LIN {X 0,Y 322.233,Z 308.252,A -85,B 0,C 180,E1 -15231.418,E2 -15231.418} C_VEL
LIN {X 0,Y 320.023,Z 295.091,A -85,B 0,C 180,E1 -15232.163,E2 -15232.163} C_VEL
LIN {X 0,Y 319.208,Z 290.536,A -85,B 0,C 180,E1 -15232.374,E2 -15232.374} C_VEL
LIN {X 0,Y 320.063,Z 282.576,A -85,B 0,C 180,E1 -15236.755,E2 -15236.755} C_VEL
LIN {X 0,Y 320.805,Z 276.273,A -85,B 0,C 180,E1 -15240.258,E2 -15240.258} C_VEL
LIN {X 0,Y 321.536,Z 271.227,A -85,B 0,C 180,E1 -15243.125,E2 -15243.125} C_VEL
LIN {X 0,Y 322.172,Z 265.933,A -85,B 0,C 180,E1 -15246.183,E2 -15246.183} C_VEL
LIN {X 0,Y 322.072,Z 262.608,A -85,B 0,C 180,E1 -15248.227,E2 -15248.227} C_VEL
LIN {X 0,Y 321.115,Z 257.021,A -85,B 0,C 180,E1 -15251.915,E2 -15251.915} C_VEL
LIN {X 0,Y 320.167,Z 252.13,A -85,B 0,C 180,E1 -15255.377,E2 -15255.377} C_VEL
LIN {X 0,Y 319.542,Z 248.686,A -85,B 0,C 180,E1 -15258.137,E2 -15258.137} C_VEL
LIN {X 0,Y 319.55,Z 248.68,A -85,B 0,C 180,E1 -15261.989,E2 -15261.989} C_VEL
LIN {X 0,Y 319.567,Z 248.677,A -85,B 0,C 180,E1 -15265.124,E2 -15265.124} C_VEL
LIN {X 0,Y 319.531,Z 248.683,A -85,B 0,C 180,E1 -15268.138,E2 -15268.138} C_VEL
LIN {X 0,Y 319.6,Z 248.671,A -85,B 0,C 180,E1 -15271.597,E2 -15271.597} C_VEL
LIN {X 0,Y 319.592,Z 248.672,A -85,B 0,C 180,E1 -15275.303,E2 -15275.303} C_VEL
LIN {X 0,Y 319.577,Z 248.679,A -85,B 0,C 180,E1 -15278.046,E2 -15278.046} C_VEL
LIN {X 0,Y 319.613,Z 248.675,A -85,B 0,C 180,E1 -15282.071,E2 -15282.071} C_VEL
LIN {X 0,Y 319.717,Z 248.663,A -85,B 0,C 180,E1 -15286.007,E2 -15286.007} C_VEL
LIN {X 0,Y 319.742,Z 248.66,A -85,B 0,C 180,E1 -15289.872,E2 -15289.872} C_VEL
LIN {X 0,Y 319.943,Z 248.634,A -85,B 0,C 180,E1 -15293.694,E2 -15293.694} C_VEL
LIN {X 0,Y 319.996,Z 248.626,A -85,B 0,C 180,E1 -15297.483,E2 -15297.483} C_VEL
LIN {X 0,Y 320.119,Z 248.607,A -85,B 0,C 180,E1 -15300,E2 -15300} C_VEL
LIN {X 0,Y 319.969,Z 248.626,A -85,B 0,C 180,E1 -15302.518,E2 -15302.518} C_VEL
LIN {X 0,Y 319.888,Z 248.635,A -85,B 0,C 180,E1 -15306.489,E2 -15306.489} C_VEL
LIN {X 0,Y 319.743,Z 248.653,A -85,B 0,C 180,E1 -15310.128,E2 -15310.128} C_VEL
LIN {X 0,Y 319.741,Z 248.653,A -85,B 0,C 180,E1 -15313.992,E2 -15313.992} C_VEL
LIN {X 0,Y 319.633,Z 248.667,A -85,B 0,C 180,E1 -15317.929,E2 -15317.929} C_VEL
LIN {X 0,Y 319.573,Z 248.675,A -85,B 0,C 180,E1 -15321.954,E2 -15321.954} C_VEL
LIN {X 0,Y 319.557,Z 248.677,A -85,B 0,C 180,E1 -15326.095,E2 -15326.095} C_VEL
LIN {X 0,Y 319.538,Z 248.682,A -85,B 0,C 180,E1 -15328.939,E2 -15328.939} C_VEL
LIN {X 0,Y 319.532,Z 248.68,A -85,B 0,C 180,E1 -15331.862,E2 -15331.862} C_VEL
LIN {X 0,Y 319.587,Z 248.673,A -85,B 0,C 180,E1 -15335.542,E2 -15335.542} C_VEL
LIN {X 0,Y 319.565,Z 248.678,A -85,B 0,C 180,E1 -15338.01,E2 -15338.01} C_VEL
LIN {X 0,Y 319.533,Z 248.68,A -85,B 0,C 180,E1 -15341.596,E2 -15341.596} C_VEL
LIN {X 0,Y 319.494,Z 248.685,A -85,B 0,C 180,E1 -15345.256,E2 -15345.256} C_VEL
LIN {X 0,Y 319.51,Z 248.686,A -85,B 0,C 180,E1 -15348.407,E2 -15348.407} C_VEL
LIN {X 0,Y 319.548,Z 248.68,A -85,B 0,C 180,E1 -15352.352,E2 -15352.352} C_VEL
LIN {X 0,Y 319.563,Z 248.677,A -85,B 0,C 180,E1 -15355.122,E2 -15355.122} C_VEL
LIN {X 0,Y 319.44,Z 248.692,A -85,B 0,C 180,E1 -15358.126,E2 -15358.126} C_VEL
LIN {X 0,Y 319.119,Z 248.735,A -85,B 0,C 180,E1 -15361.755,E2 -15361.755} C_VEL
LIN {X 0,Y 319.035,Z 248.746,A -85,B 0,C 180,E1 -15362.443,E2 -15362.443} C_VEL
LIN {X 0,Y 318.918,Z 251.041,A -85,B 0,C 180,E1 -15365.245,E2 -15365.245} C_VEL
LIN {X 0,Y 318.771,Z 254.574,A -85,B 0,C 180,E1 -15369.342,E2 -15369.342} C_VEL
LIN {X 0,Y 318.715,Z 256.98,A -85,B 0,C 180,E1 -15371.993,E2 -15371.993} C_VEL
LIN {X 0,Y 322.509,Z 270.16,A -85,B 0,C 180,E1 -15372.833,E2 -15372.833} C_VEL
LIN {X 0,Y 325.314,Z 281.932,A -85,B 0,C 180,E1 -15373.777,E2 -15373.777} C_VEL
LIN {X 0,Y 326.484,Z 288.024,A -85,B 0,C 180,E1 -15374.34,E2 -15374.34} C_VEL
LIN {X 0,Y 325.488,Z 299.937,A -85,B 0,C 180,E1 -15375.461,E2 -15375.461} C_VEL
LIN {X 0,Y 324.31,Z 311.411,A -85,B 0,C 180,E1 -15376.846,E2 -15376.846} C_VEL
LIN {X 0,Y 323.016,Z 321.596,A -85,B 0,C 180,E1 -15378.388,E2 -15378.388} C_VEL
LIN {X 0,Y 321.817,Z 329.869,A -85,B 0,C 180,E1 -15379.937,E2 -15379.937} C_VEL
LIN {X 0,Y 321.08,Z 336.714,A -85,B 0,C 180,E1 -15381.502,E2 -15381.502} C_VEL
LIN {X 0,Y 320.196,Z 342.455,A -85,B 0,C 180,E1 -15383.065,E2 -15383.065} C_VEL
LIN {X 0,Y 319.336,Z 348.048,A -85,B 0,C 180,E1 -15384.948,E2 -15384.948} C_VEL
LIN {X 0,Y 318.76,Z 352.451,A -85,B 0,C 180,E1 -15386.838,E2 -15386.838} C_VEL
LIN {X 0,Y 318.368,Z 355.798,A -85,B 0,C 180,E1 -15388.733,E2 -15388.733} C_VEL
LIN {X 0,Y 318.217,Z 358.723,A -85,B 0,C 180,E1 -15391.264,E2 -15391.264} C_VEL
LIN {X 0,Y 318.127,Z 359.61,A -85,B 0,C 180,E1 -15392.53,E2 -15392.53} C_VEL
LIN {X 0,Y 318.094,Z 360.081,A -85,B 0,C 180,E1 -15393.799,E2 -15393.799} C_VEL
LIN {X 0,Y 318.194,Z 360.147,A -85,B 0,C 180,E1 -15395.067,E2 -15395.067} C_VEL
LIN {X 0,Y 318.364,Z 359.155,A -85,B 0,C 180,E1 -15397.609,E2 -15397.609} C_VEL
LIN {X 0,Y 318.488,Z 358.053,A -85,B 0,C 180,E1 -15398.884,E2 -15398.884} C_VEL
LIN {X 0,Y 318.747,Z 356.52,A -85,B 0,C 180,E1 -15400.158,E2 -15400.158} C_VEL
LIN {X 0,Y 319.241,Z 353.431,A -85,B 0,C 180,E1 -15402.07,E2 -15402.07} C_VEL
LIN {X 0,Y 320.046,Z 349.274,A -85,B 0,C 180,E1 -15403.976,E2 -15403.976} C_VEL
LIN {X 0,Y 321.153,Z 343.03,A -85,B 0,C 180,E1 -15406.167,E2 -15406.167} C_VEL
LIN {X 0,Y 322.429,Z 335.97,A -85,B 0,C 180,E1 -15408.094,E2 -15408.094} C_VEL
LIN {X 0,Y 323.916,Z 327.221,A -85,B 0,C 180,E1 -15409.98,E2 -15409.98} C_VEL
LIN {X 0,Y 325.428,Z 317.221,A -85,B 0,C 180,E1 -15411.708,E2 -15411.708} C_VEL
LIN {X 0,Y 326.945,Z 307.014,A -85,B 0,C 180,E1 -15413.096,E2 -15413.096} C_VEL
LIN {X 0,Y 328.403,Z 295.417,A -85,B 0,C 180,E1 -15414.347,E2 -15414.347} C_VEL
LIN {X 0,Y 328.672,Z 291.825,A -85,B 0,C 180,E1 -15414.684,E2 -15414.684} C_VEL
LIN {X 0,Y 326.402,Z 281.122,A -85,B 0,C 180,E1 -15415.775,E2 -15415.775} C_VEL
LIN {X 0,Y 322.82,Z 268.661,A -85,B 0,C 180,E1 -15416.868,E2 -15416.868} C_VEL
LIN {X 0,Y 318.979,Z 257.353,A -85,B 0,C 180,E1 -15417.719,E2 -15417.719} C_VEL
LIN {X 0,Y 319.063,Z 254.737,A -85,B 0,C 180,E1 -15420.789,E2 -15420.789} C_VEL
LIN {X 0,Y 319.183,Z 252.598,A -85,B 0,C 180,E1 -15423.397,E2 -15423.397} C_VEL
LIN {X 0,Y 319.318,Z 250.168,A -85,B 0,C 180,E1 -15426.457,E2 -15426.457} C_VEL
LIN {X 0,Y 319.346,Z 248.967,A -85,B 0,C 180,E1 -15428.037,E2 -15428.037} C_VEL
LIN {X 0,Y 319.465,Z 248.691,A -85,B 0,C 180,E1 -15429.648,E2 -15429.648} C_VEL
LIN {X 0,Y 319.513,Z 248.686,A -85,B 0,C 180,E1 -15433.458,E2 -15433.458} C_VEL
LIN {X 0,Y 319.546,Z 248.682,A -85,B 0,C 180,E1 -15437.015,E2 -15437.015} C_VEL
LIN {X 0,Y 319.539,Z 248.683,A -85,B 0,C 180,E1 -15440.369,E2 -15440.369} C_VEL
LIN {X 0,Y 319.551,Z 248.677,A -85,B 0,C 180,E1 -15443.571,E2 -15443.571} C_VEL
LIN {X 0,Y 319.568,Z 248.677,A -85,B 0,C 180,E1 -15446.685,E2 -15446.685} C_VEL
LIN {X 0,Y 319.575,Z 248.676,A -85,B 0,C 180,E1 -15449.615,E2 -15449.615} C_VEL
LIN {X 0,Y 319.596,Z 248.671,A -85,B 0,C 180,E1 -15452.497,E2 -15452.497} C_VEL
LIN {X 0,Y 319.621,Z 248.673,A -85,B 0,C 180,E1 -15454.409,E2 -15454.409} C_VEL
LIN {X 0,Y 318.898,Z 248.762,A -85,B 0,C 180,E1 -15455.46,E2 -15455.46} C_VEL
LIN {X 0,Y 316.002,Z 249.124,A -85,B 0,C 180,E1 -15457.171,E2 -15457.171} C_VEL
LIN {X 0,Y 313.605,Z 249.421,A -85,B 0,C 180,E1 -15458.558,E2 -15458.558} C_VEL
LIN {X 0,Y 312.617,Z 249.543,A -85,B 0,C 180,E1 -15459.632,E2 -15459.632} C_VEL
LIN {X 0,Y 312.557,Z 249.55,A -85,B 0,C 180,E1 -15459.995,E2 -15459.995} C_VEL
LIN {X 0,Y 312.596,Z 249.547,A -85,B 0,C 180,E1 -15463.006,E2 -15463.006} C_VEL
LIN {X 0,Y 312.683,Z 249.537,A -85,B 0,C 180,E1 -15465.685,E2 -15465.685} C_VEL
LIN {X 0,Y 312.69,Z 249.535,A -85,B 0,C 180,E1 -15469.641,E2 -15469.641} C_VEL
LIN {X 0,Y 312.864,Z 249.516,A -85,B 0,C 180,E1 -15472.254,E2 -15472.254} C_VEL
LIN {X 0,Y 312.713,Z 249.532,A -85,B 0,C 180,E1 -15474.842,E2 -15474.842} C_VEL
LIN {X 0,Y 312.943,Z 249.504,A -85,B 0,C 180,E1 -15477.425,E2 -15477.425} C_VEL
LIN {X 0,Y 313.072,Z 249.488,A -85,B 0,C 180,E1 -15480,E2 -15480} C_VEL
LIN {X 0,Y 312.928,Z 249.506,A -85,B 0,C 180,E1 -15482.574,E2 -15482.574} C_VEL
LIN {X 0,Y 312.902,Z 249.508,A -85,B 0,C 180,E1 -15486.448,E2 -15486.448} C_VEL
LIN {X 0,Y 312.776,Z 249.525,A -85,B 0,C 180,E1 -15489.049,E2 -15489.049} C_VEL
LIN {X 0,Y 312.622,Z 249.541,A -85,B 0,C 180,E1 -15492.991,E2 -15492.991} C_VEL
LIN {X 0,Y 312.627,Z 249.537,A -85,B 0,C 180,E1 -15495.65,E2 -15495.65} C_VEL
LIN {X 0,Y 312.62,Z 249.539,A -85,B 0,C 180,E1 -15499.237,E2 -15499.237} C_VEL
LIN {X 0,Y 312.535,Z 249.554,A -85,B 0,C 180,E1 -15502.79,E2 -15502.79} C_VEL
LIN {X 0,Y 312.592,Z 249.547,A -85,B 0,C 180,E1 -15505.937,E2 -15505.937} C_VEL
LIN {X 0,Y 312.54,Z 249.555,A -85,B 0,C 180,E1 -15509.65,E2 -15509.65} C_VEL
LIN {X 0,Y 312.51,Z 249.558,A -85,B 0,C 180,E1 -15513.69,E2 -15513.69} C_VEL
LIN {X 0,Y 312.516,Z 249.554,A -85,B 0,C 180,E1 -15517.386,E2 -15517.386} C_VEL
LIN {X 0,Y 312.563,Z 249.741,A -85,B 0,C 180,E1 -15519.019,E2 -15519.019} C_VEL
LIN {X 0,Y 313.397,Z 254.62,A -85,B 0,C 180,E1 -15523.155,E2 -15523.155} C_VEL
LIN {X 0,Y 314.118,Z 258.292,A -85,B 0,C 180,E1 -15526.088,E2 -15526.088} C_VEL
LIN {X 0,Y 315.018,Z 263.182,A -85,B 0,C 180,E1 -15529.688,E2 -15529.688} C_VEL
LIN {X 0,Y 315.532,Z 266.879,A -85,B 0,C 180,E1 -15532.231,E2 -15532.231} C_VEL
LIN {X 0,Y 315.459,Z 269.519,A -85,B 0,C 180,E1 -15533.947,E2 -15533.947} C_VEL
LIN {X 0,Y 314.733,Z 274.207,A -85,B 0,C 180,E1 -15536.835,E2 -15536.835} C_VEL
LIN {X 0,Y 313.649,Z 281.043,A -85,B 0,C 180,E1 -15540.913,E2 -15540.913} C_VEL
LIN {X 0,Y 312.764,Z 287.604,A -85,B 0,C 180,E1 -15544.729,E2 -15544.729} C_VEL
LIN {X 0,Y 312.495,Z 289.833,A -85,B 0,C 180,E1 -15546.012,E2 -15546.012} C_VEL
LIN {X 0,Y 315.709,Z 304.105,A -85,B 0,C 180,E1 -15546.896,E2 -15546.896} C_VEL
LIN {X 0,Y 317.8,Z 317.281,A -85,B 0,C 180,E1 -15547.919,E2 -15547.919} C_VEL
LIN {X 0,Y 318.738,Z 328.567,A -85,B 0,C 180,E1 -15548.969,E2 -15548.969} C_VEL
LIN {X 0,Y 318.968,Z 338.241,A -85,B 0,C 180,E1 -15550.033,E2 -15550.033} C_VEL
LIN {X 0,Y 317.255,Z 349.546,A -85,B 0,C 180,E1 -15551.433,E2 -15551.433} C_VEL
LIN {X 0,Y 315.816,Z 358.663,A -85,B 0,C 180,E1 -15552.853,E2 -15552.853} C_VEL
LIN {X 0,Y 314.305,Z 368.534,A -85,B 0,C 180,E1 -15554.77,E2 -15554.77} C_VEL
LIN {X 0,Y 313.094,Z 376.489,A -85,B 0,C 180,E1 -15556.7,E2 -15556.7} C_VEL
LIN {X 0,Y 312.179,Z 381.882,A -85,B 0,C 180,E1 -15558.312,E2 -15558.312} C_VEL
LIN {X 0,Y 311.522,Z 387.187,A -85,B 0,C 180,E1 -15560.261,E2 -15560.261} C_VEL
LIN {X 0,Y 311.062,Z 391.324,A -85,B 0,C 180,E1 -15562.211,E2 -15562.211} C_VEL
LIN {X 0,Y 310.898,Z 394.279,A -85,B 0,C 180,E1 -15564.066,E2 -15564.066} C_VEL
LIN {X 0,Y 310.842,Z 396.536,A -85,B 0,C 180,E1 -15566.113,E2 -15566.113} C_VEL
LIN {X 0,Y 310.775,Z 397.451,A -85,B 0,C 180,E1 -15567.41,E2 -15567.41} C_VEL
LIN {X 0,Y 310.847,Z 397.944,A -85,B 0,C 180,E1 -15568.706,E2 -15568.706} C_VEL
LIN {X 0,Y 310.959,Z 398.025,A -85,B 0,C 180,E1 -15570.002,E2 -15570.002} C_VEL
LIN {X 0,Y 310.885,Z 397.703,A -85,B 0,C 180,E1 -15571.297,E2 -15571.297} C_VEL
LIN {X 0,Y 310.798,Z 396.988,A -85,B 0,C 180,E1 -15572.594,E2 -15572.594} C_VEL
LIN {X 0,Y 310.849,Z 395.854,A -85,B 0,C 180,E1 -15573.891,E2 -15573.891} C_VEL
LIN {X 0,Y 310.908,Z 393.171,A -85,B 0,C 180,E1 -15575.95,E2 -15575.95} C_VEL
LIN {X 0,Y 311.222,Z 388.384,A -85,B 0,C 180,E1 -15578.442,E2 -15578.442} C_VEL
LIN {X 0,Y 311.718,Z 383.36,A -85,B 0,C 180,E1 -15580.393,E2 -15580.393} C_VEL
LIN {X 0,Y 312.456,Z 377.046,A -85,B 0,C 180,E1 -15582.34,E2 -15582.34} C_VEL
LIN {X 0,Y 313.521,Z 369.157,A -85,B 0,C 180,E1 -15584.277,E2 -15584.277} C_VEL
LIN {X 0,Y 314.779,Z 359.909,A -85,B 0,C 180,E1 -15586.095,E2 -15586.095} C_VEL
LIN {X 0,Y 315.995,Z 350.191,A -85,B 0,C 180,E1 -15587.642,E2 -15587.642} C_VEL
LIN {X 0,Y 317.503,Z 338.943,A -85,B 0,C 180,E1 -15589.058,E2 -15589.058} C_VEL
LIN {X 0,Y 317.917,Z 334.534,A -85,B 0,C 180,E1 -15589.535,E2 -15589.535} C_VEL
LIN {X 0,Y 316.857,Z 321.893,A -85,B 0,C 180,E1 -15590.788,E2 -15590.788} C_VEL
LIN {X 0,Y 315.383,Z 308.783,A -85,B 0,C 180,E1 -15591.811,E2 -15591.811} C_VEL
LIN {X 0,Y 313.189,Z 295.309,A -85,B 0,C 180,E1 -15592.605,E2 -15592.605} C_VEL
LIN {X 0,Y 312.208,Z 290.074,A -85,B 0,C 180,E1 -15592.887,E2 -15592.887} C_VEL
LIN {X 0,Y 312.964,Z 283.358,A -85,B 0,C 180,E1 -15596.689,E2 -15596.689} C_VEL
LIN {X 0,Y 313.749,Z 277.065,A -85,B 0,C 180,E1 -15600.267,E2 -15600.267} C_VEL
LIN {X 0,Y 314.516,Z 272.064,A -85,B 0,C 180,E1 -15603.195,E2 -15603.195} C_VEL
LIN {X 0,Y 315.029,Z 268.249,A -85,B 0,C 180,E1 -15605.455,E2 -15605.455} C_VEL
LIN {X 0,Y 315.124,Z 264.401,A -85,B 0,C 180,E1 -15607.822,E2 -15607.822} C_VEL
LIN {X 0,Y 314.294,Z 259.222,A -85,B 0,C 180,E1 -15611.288,E2 -15611.288} C_VEL
LIN {X 0,Y 313.314,Z 253.955,A -85,B 0,C 180,E1 -15615.043,E2 -15615.043} C_VEL
LIN {X 0,Y 312.494,Z 249.563,A -85,B 0,C 180,E1 -15618.585,E2 -15618.585} C_VEL
LIN {X 0,Y 312.527,Z 249.558,A -85,B 0,C 180,E1 -15622.615,E2 -15622.615} C_VEL
LIN {X 0,Y 312.527,Z 249.557,A -85,B 0,C 180,E1 -15626.312,E2 -15626.312} C_VEL
LIN {X 0,Y 312.51,Z 249.559,A -85,B 0,C 180,E1 -15630.346,E2 -15630.346} C_VEL
LIN {X 0,Y 312.545,Z 249.554,A -85,B 0,C 180,E1 -15634.09,E2 -15634.09} C_VEL
LIN {X 0,Y 312.574,Z 249.548,A -85,B 0,C 180,E1 -15637.528,E2 -15637.528} C_VEL
LIN {X 0,Y 312.57,Z 249.549,A -85,B 0,C 180,E1 -15641.652,E2 -15641.652} C_VEL
LIN {X 0,Y 312.659,Z 249.54,A -85,B 0,C 180,E1 -15645.685,E2 -15645.685} C_VEL
LIN {X 0,Y 312.692,Z 249.536,A -85,B 0,C 180,E1 -15649.642,E2 -15649.642} C_VEL
LIN {X 0,Y 312.899,Z 249.51,A -85,B 0,C 180,E1 -15653.552,E2 -15653.552} C_VEL
LIN {X 0,Y 312.943,Z 249.504,A -85,B 0,C 180,E1 -15657.426,E2 -15657.426} C_VEL
LIN {X 0,Y 313.074,Z 249.485,A -85,B 0,C 180,E1 -15660,E2 -15660} C_VEL
LIN {X 0,Y 312.917,Z 249.504,A -85,B 0,C 180,E1 -15662.575,E2 -15662.575} C_VEL
LIN {X 0,Y 312.844,Z 249.513,A -85,B 0,C 180,E1 -15666.468,E2 -15666.468} C_VEL
LIN {X 0,Y 312.759,Z 249.527,A -85,B 0,C 180,E1 -15669.05,E2 -15669.05} C_VEL
LIN {X 0,Y 312.643,Z 249.542,A -85,B 0,C 180,E1 -15672.991,E2 -15672.991} C_VEL
LIN {X 0,Y 312.63,Z 249.54,A -85,B 0,C 180,E1 -15675.65,E2 -15675.65} C_VEL
LIN {X 0,Y 312.567,Z 249.546,A -85,B 0,C 180,E1 -15679.711,E2 -15679.711} C_VEL
LIN {X 0,Y 312.523,Z 249.558,A -85,B 0,C 180,E1 -15682.775,E2 -15682.775} C_VEL
LIN {X 0,Y 312.49,Z 249.562,A -85,B 0,C 180,E1 -15686.732,E2 -15686.732} C_VEL
LIN {X 0,Y 312.48,Z 249.558,A -85,B 0,C 180,E1 -15689.657,E2 -15689.657} C_VEL
LIN {X 0,Y 312.528,Z 249.552,A -85,B 0,C 180,E1 -15693.688,E2 -15693.688} C_VEL
LIN {X 0,Y 312.533,Z 249.551,A -85,B 0,C 180,E1 -15697.384,E2 -15697.384} C_VEL
LIN {X 0,Y 312.498,Z 249.558,A -85,B 0,C 180,E1 -15700.708,E2 -15700.708} C_VEL
LIN {X 0,Y 312.458,Z 249.566,A -85,B 0,C 180,E1 -15704.209,E2 -15704.209} C_VEL
LIN {X 0,Y 312.461,Z 249.565,A -85,B 0,C 180,E1 -15707.924,E2 -15707.924} C_VEL
LIN {X 0,Y 312.483,Z 249.563,A -85,B 0,C 180,E1 -15711.923,E2 -15711.923} C_VEL
LIN {X 0,Y 312.536,Z 249.554,A -85,B 0,C 180,E1 -15714.219,E2 -15714.219} C_VEL
LIN {X 0,Y 312.457,Z 249.562,A -85,B 0,C 180,E1 -15717.326,E2 -15717.326} C_VEL
LIN {X 0,Y 312.208,Z 249.592,A -85,B 0,C 180,E1 -15720.313,E2 -15720.313} C_VEL
LIN {X 0,Y 312.077,Z 249.612,A -85,B 0,C 180,E1 -15721.774,E2 -15721.774} C_VEL
LIN {X 0,Y 311.931,Z 250.276,A -85,B 0,C 180,E1 -15723.215,E2 -15723.215} C_VEL
LIN {X 0,Y 311.818,Z 252.66,A -85,B 0,C 180,E1 -15726.063,E2 -15726.063} C_VEL
LIN {X 0,Y 311.679,Z 256.256,A -85,B 0,C 180,E1 -15730.229,E2 -15730.229} C_VEL
LIN {X 0,Y 311.68,Z 257.388,A -85,B 0,C 180,E1 -15731.485,E2 -15731.485} C_VEL
LIN {X 0,Y 316.082,Z 272.613,A -85,B 0,C 180,E1 -15732.531,E2 -15732.531} C_VEL
LIN {X 0,Y 318.751,Z 284.177,A -85,B 0,C 180,E1 -15733.516,E2 -15733.516} C_VEL
LIN {X 0,Y 319.685,Z 289.06,A -85,B 0,C 180,E1 -15733.993,E2 -15733.993} C_VEL
LIN {X 0,Y 318.671,Z 300.858,A -85,B 0,C 180,E1 -15735.143,E2 -15735.143} C_VEL
LIN {X 0,Y 317.444,Z 312.246,A -85,B 0,C 180,E1 -15736.556,E2 -15736.556} C_VEL
LIN {X 0,Y 316.128,Z 322.157,A -85,B 0,C 180,E1 -15738.099,E2 -15738.099} C_VEL
LIN {X 0,Y 314.873,Z 330.553,A -85,B 0,C 180,E1 -15739.712,E2 -15739.712} C_VEL
LIN {X 0,Y 314.101,Z 337.354,A -85,B 0,C 180,E1 -15741.311,E2 -15741.311} C_VEL
LIN {X 0,Y 313.199,Z 343.057,A -85,B 0,C 180,E1 -15742.909,E2 -15742.909} C_VEL
LIN {X 0,Y 312.311,Z 348.613,A -85,B 0,C 180,E1 -15744.834,E2 -15744.834} C_VEL
LIN {X 0,Y 311.701,Z 352.985,A -85,B 0,C 180,E1 -15746.767,E2 -15746.767} C_VEL
LIN {X 0,Y 311.308,Z 356.301,A -85,B 0,C 180,E1 -15748.705,E2 -15748.705} C_VEL
LIN {X 0,Y 311.139,Z 359.198,A -85,B 0,C 180,E1 -15751.292,E2 -15751.292} C_VEL
LIN {X 0,Y 311.036,Z 360.071,A -85,B 0,C 180,E1 -15752.588,E2 -15752.588} C_VEL
LIN {X 0,Y 311.114,Z 360.567,A -85,B 0,C 180,E1 -15755.182,E2 -15755.182} C_VEL
LIN {X 0,Y 311.308,Z 359.548,A -85,B 0,C 180,E1 -15757.783,E2 -15757.783} C_VEL
LIN {X 0,Y 311.457,Z 358.418,A -85,B 0,C 180,E1 -15759.086,E2 -15759.086} C_VEL
LIN {X 0,Y 311.737,Z 356.87,A -85,B 0,C 180,E1 -15760.389,E2 -15760.389} C_VEL
LIN {X 0,Y 312.274,Z 353.751,A -85,B 0,C 180,E1 -15762.343,E2 -15762.343} C_VEL
LIN {X 0,Y 313.104,Z 349.562,A -85,B 0,C 180,E1 -15764.293,E2 -15764.293} C_VEL
LIN {X 0,Y 314.32,Z 343.182,A -85,B 0,C 180,E1 -15766.562,E2 -15766.562} C_VEL
LIN {X 0,Y 315.635,Z 336.162,A -85,B 0,C 180,E1 -15768.497,E2 -15768.497} C_VEL
LIN {X 0,Y 317.221,Z 327.363,A -85,B 0,C 180,E1 -15770.42,E2 -15770.42} C_VEL
LIN {X 0,Y 318.627,Z 318.317,A -85,B 0,C 180,E1 -15772.02,E2 -15772.02} C_VEL
LIN {X 0,Y 320.223,Z 308.281,A -85,B 0,C 180,E1 -15773.438,E2 -15773.438} C_VEL
LIN {X 0,Y 321.741,Z 296.711,A -85,B 0,C 180,E1 -15774.731,E2 -15774.731} C_VEL
LIN {X 0,Y 321.945,Z 292.622,A -85,B 0,C 180,E1 -15775.139,E2 -15775.139} C_VEL
LIN {X 0,Y 319.618,Z 281.915,A -85,B 0,C 180,E1 -15776.273,E2 -15776.273} C_VEL
LIN {X 0,Y 316.113,Z 269.833,A -85,B 0,C 180,E1 -15777.378,E2 -15777.378} C_VEL
LIN {X 0,Y 311.988,Z 258.227,A -85,B 0,C 180,E1 -15778.278,E2 -15778.278} C_VEL
LIN {X 0,Y 311.934,Z 257.819,A -85,B 0,C 180,E1 -15778.306,E2 -15778.306} C_VEL
LIN {X 0,Y 312.062,Z 255.405,A -85,B 0,C 180,E1 -15781.195,E2 -15781.195} C_VEL
LIN {X 0,Y 312.169,Z 252.919,A -85,B 0,C 180,E1 -15784.25,E2 -15784.25} C_VEL
LIN {X 0,Y 312.354,Z 250.031,A -85,B 0,C 180,E1 -15788.046,E2 -15788.046} C_VEL
LIN {X 0,Y 312.346,Z 249.577,A -85,B 0,C 180,E1 -15789.049,E2 -15789.049} C_VEL
LIN {X 0,Y 312.456,Z 249.565,A -85,B 0,C 180,E1 -15792.434,E2 -15792.434} C_VEL
LIN {X 0,Y 312.451,Z 249.566,A -85,B 0,C 180,E1 -15796.033,E2 -15796.033} C_VEL
LIN {X 0,Y 312.496,Z 249.56,A -85,B 0,C 180,E1 -15799.873,E2 -15799.873} C_VEL
LIN {X 0,Y 312.53,Z 249.556,A -85,B 0,C 180,E1 -15802.615,E2 -15802.615} C_VEL
LIN {X 0,Y 312.511,Z 249.555,A -85,B 0,C 180,E1 -15806.31,E2 -15806.31} C_VEL
LIN {X 0,Y 312.529,Z 249.554,A -85,B 0,C 180,E1 -15810.348,E2 -15810.348} C_VEL
LIN {X 0,Y 312.579,Z 249.549,A -85,B 0,C 180,E1 -15814.403,E2 -15814.403} C_VEL
LIN {X 0,Y 312.577,Z 249.55,A -85,B 0,C 180,E1 -15817.528,E2 -15817.528} C_VEL
LIN {X 0,Y 312.557,Z 249.55,A -85,B 0,C 180,E1 -15819.995,E2 -15819.995} C_VEL
LIN {X 0,Y 311.961,Z 249.628,A -85,B 0,C 180,E1 -15821.071,E2 -15821.071} C_VEL
LIN {X 0,Y 309.19,Z 249.977,A -85,B 0,C 180,E1 -15822.823,E2 -15822.823} C_VEL
LIN {X 0,Y 306.782,Z 250.275,A -85,B 0,C 180,E1 -15824.243,E2 -15824.243} C_VEL
LIN {X 0,Y 305.71,Z 250.406,A -85,B 0,C 180,E1 -15825.342,E2 -15825.342} C_VEL
LIN {X 0,Y 305.605,Z 250.416,A -85,B 0,C 180,E1 -15825.715,E2 -15825.715} C_VEL
LIN {X 0,Y 305.627,Z 250.416,A -85,B 0,C 180,E1 -15829.399,E2 -15829.399} C_VEL
LIN {X 0,Y 305.805,Z 250.395,A -85,B 0,C 180,E1 -15832.074,E2 -15832.074} C_VEL
LIN {X 0,Y 305.684,Z 250.408,A -85,B 0,C 180,E1 -15834.723,E2 -15834.723} C_VEL
LIN {X 0,Y 305.947,Z 250.377,A -85,B 0,C 180,E1 -15838.684,E2 -15838.684} C_VEL
LIN {X 0,Y 305.944,Z 250.376,A -85,B 0,C 180,E1 -15841.316,E2 -15841.316} C_VEL
LIN {X 0,Y 305.682,Z 250.409,A -85,B 0,C 180,E1 -15845.277,E2 -15845.277} C_VEL
LIN {X 0,Y 305.804,Z 250.393,A -85,B 0,C 180,E1 -15847.926,E2 -15847.926} C_VEL
LIN {X 0,Y 305.592,Z 250.421,A -85,B 0,C 180,E1 -15851.945,E2 -15851.945} C_VEL
LIN {X 0,Y 305.626,Z 250.41,A -85,B 0,C 180,E1 -15855.035,E2 -15855.035} C_VEL
LIN {X 0,Y 305.566,Z 250.418,A -85,B 0,C 180,E1 -15859.446,E2 -15859.446} C_VEL
LIN {X 0,Y 305.48,Z 250.433,A -85,B 0,C 180,E1 -15863.042,E2 -15863.042} C_VEL
LIN {X 0,Y 305.537,Z 250.426,A -85,B 0,C 180,E1 -15866.228,E2 -15866.228} C_VEL
LIN {X 0,Y 305.494,Z 250.432,A -85,B 0,C 180,E1 -15869.054,E2 -15869.054} C_VEL
LIN {X 0,Y 305.456,Z 250.437,A -85,B 0,C 180,E1 -15873.518,E2 -15873.518} C_VEL
LIN {X 0,Y 305.486,Z 250.43,A -85,B 0,C 180,E1 -15877.565,E2 -15877.565} C_VEL
LIN {X 0,Y 305.543,Z 250.673,A -85,B 0,C 180,E1 -15878.393,E2 -15878.393} C_VEL
LIN {X 0,Y 306.361,Z 255.637,A -85,B 0,C 180,E1 -15882.773,E2 -15882.773} C_VEL
LIN {X 0,Y 307.295,Z 260.472,A -85,B 0,C 180,E1 -15886.68,E2 -15886.68} C_VEL
LIN {X 0,Y 308.188,Z 265.372,A -85,B 0,C 180,E1 -15890.321,E2 -15890.321} C_VEL
LIN {X 0,Y 308.567,Z 269.02,A -85,B 0,C 180,E1 -15892.861,E2 -15892.861} C_VEL
LIN {X 0,Y 308.171,Z 272.701,A -85,B 0,C 180,E1 -15895.243,E2 -15895.243} C_VEL
LIN {X 0,Y 307.055,Z 278.764,A -85,B 0,C 180,E1 -15899.006,E2 -15899.006} C_VEL
LIN {X 0,Y 306.196,Z 284.842,A -85,B 0,C 180,E1 -15902.676,E2 -15902.676} C_VEL
LIN {X 0,Y 305.559,Z 289.397,A -85,B 0,C 180,E1 -15905.387,E2 -15905.387} C_VEL
LIN {X 0,Y 308.795,Z 303.555,A -85,B 0,C 180,E1 -15906.295,E2 -15906.295} C_VEL
LIN {X 0,Y 310.851,Z 316.291,A -85,B 0,C 180,E1 -15907.311,E2 -15907.311} C_VEL
LIN {X 0,Y 311.888,Z 327.451,A -85,B 0,C 180,E1 -15908.374,E2 -15908.374} C_VEL
LIN {X 0,Y 312.262,Z 338.159,A -85,B 0,C 180,E1 -15909.585,E2 -15909.585} C_VEL
LIN {X 0,Y 310.516,Z 349.379,A -85,B 0,C 180,E1 -15911.015,E2 -15911.015} C_VEL
LIN {X 0,Y 309.015,Z 358.449,A -85,B 0,C 180,E1 -15912.464,E2 -15912.464} C_VEL
LIN {X 0,Y 307.715,Z 366.79,A -85,B 0,C 180,E1 -15914.095,E2 -15914.095} C_VEL
LIN {X 0,Y 306.353,Z 374.972,A -85,B 0,C 180,E1 -15916.064,E2 -15916.064} C_VEL
LIN {X 0,Y 305.189,Z 381.572,A -85,B 0,C 180,E1 -15918.041,E2 -15918.041} C_VEL
LIN {X 0,Y 304.481,Z 386.853,A -85,B 0,C 180,E1 -15920.033,E2 -15920.033} C_VEL
LIN {X 0,Y 304.015,Z 390.969,A -85,B 0,C 180,E1 -15922.029,E2 -15922.029} C_VEL
LIN {X 0,Y 303.819,Z 394.128,A -85,B 0,C 180,E1 -15924.091,E2 -15924.091} C_VEL
LIN {X 0,Y 303.751,Z 396.141,A -85,B 0,C 180,E1 -15926.022,E2 -15926.022} C_VEL
LIN {X 0,Y 303.698,Z 397.046,A -85,B 0,C 180,E1 -15927.349,E2 -15927.349} C_VEL
LIN {X 0,Y 303.754,Z 397.521,A -85,B 0,C 180,E1 -15928.676,E2 -15928.676} C_VEL
LIN {X 0,Y 303.871,Z 397.593,A -85,B 0,C 180,E1 -15930.002,E2 -15930.002} C_VEL
LIN {X 0,Y 303.791,Z 397.261,A -85,B 0,C 180,E1 -15931.328,E2 -15931.328} C_VEL
LIN {X 0,Y 303.719,Z 396.538,A -85,B 0,C 180,E1 -15932.655,E2 -15932.655} C_VEL
LIN {X 0,Y 303.781,Z 395.385,A -85,B 0,C 180,E1 -15933.982,E2 -15933.982} C_VEL
LIN {X 0,Y 303.84,Z 392.909,A -85,B 0,C 180,E1 -15935.947,E2 -15935.947} C_VEL
LIN {X 0,Y 304.036,Z 389.314,A -85,B 0,C 180,E1 -15937.974,E2 -15937.974} C_VEL
LIN {X 0,Y 304.48,Z 384.658,A -85,B 0,C 180,E1 -15939.971,E2 -15939.971} C_VEL
LIN {X 0,Y 305.343,Z 377.616,A -85,B 0,C 180,E1 -15942.295,E2 -15942.295} C_VEL
LIN {X 0,Y 306.416,Z 370.001,A -85,B 0,C 180,E1 -15944.276,E2 -15944.276} C_VEL
LIN {X 0,Y 307.562,Z 362.231,A -85,B 0,C 180,E1 -15945.917,E2 -15945.917} C_VEL
LIN {X 0,Y 308.786,Z 352.748,A -85,B 0,C 180,E1 -15947.554,E2 -15947.554} C_VEL
LIN {X 0,Y 310.25,Z 342.232,A -85,B 0,C 180,E1 -15949.006,E2 -15949.006} C_VEL
LIN {X 0,Y 310.999,Z 335.277,A -85,B 0,C 180,E1 -15949.816,E2 -15949.816} C_VEL
LIN {X 0,Y 310.109,Z 323.601,A -85,B 0,C 180,E1 -15951.036,E2 -15951.036} C_VEL
LIN {X 0,Y 308.7,Z 310.256,A -85,B 0,C 180,E1 -15952.141,E2 -15952.141} C_VEL
LIN {X 0,Y 306.665,Z 297.425,A -85,B 0,C 180,E1 -15952.971,E2 -15952.971} C_VEL
LIN {X 0,Y 305.206,Z 289.712,A -85,B 0,C 180,E1 -15953.361,E2 -15953.361} C_VEL
LIN {X 0,Y 306.011,Z 282.878,A -85,B 0,C 180,E1 -15957.346,E2 -15957.346} C_VEL
LIN {X 0,Y 306.831,Z 276.603,A -85,B 0,C 180,E1 -15961.024,E2 -15961.024} C_VEL
LIN {X 0,Y 307.617,Z 271.684,A -85,B 0,C 180,E1 -15964,E2 -15964} C_VEL
LIN {X 0,Y 308.094,Z 267.8,A -85,B 0,C 180,E1 -15966.379,E2 -15966.379} C_VEL
LIN {X 0,Y 308.084,Z 265.233,A -85,B 0,C 180,E1 -15968.021,E2 -15968.021} C_VEL
LIN {X 0,Y 307.225,Z 260.061,A -85,B 0,C 180,E1 -15971.562,E2 -15971.562} C_VEL
LIN {X 0,Y 306.267,Z 254.954,A -85,B 0,C 180,E1 -15975.348,E2 -15975.348} C_VEL
LIN {X 0,Y 305.454,Z 250.44,A -85,B 0,C 180,E1 -15979.002,E2 -15979.002} C_VEL
LIN {X 0,Y 305.474,Z 250.434,A -85,B 0,C 180,E1 -15981.597,E2 -15981.597} C_VEL
LIN {X 0,Y 305.469,Z 250.435,A -85,B 0,C 180,E1 -15984.888,E2 -15984.888} C_VEL
LIN {X 0,Y 305.449,Z 250.438,A -85,B 0,C 180,E1 -15988.359,E2 -15988.359} C_VEL
LIN {X 0,Y 305.497,Z 250.428,A -85,B 0,C 180,E1 -15991.112,E2 -15991.112} C_VEL
LIN {X 0,Y 305.516,Z 250.429,A -85,B 0,C 180,E1 -15994.083,E2 -15994.083} C_VEL
LIN {X 0,Y 305.483,Z 250.434,A -85,B 0,C 180,E1 -15998.402,E2 -15998.402} C_VEL
LIN {X 0,Y 305.523,Z 250.425,A -85,B 0,C 180,E1 -16001.213,E2 -16001.213} C_VEL
LIN {X 0,Y 305.587,Z 250.419,A -85,B 0,C 180,E1 -16005.346,E2 -16005.346} C_VEL
LIN {X 0,Y 305.63,Z 250.414,A -85,B 0,C 180,E1 -16009.4,E2 -16009.4} C_VEL
LIN {X 0,Y 305.78,Z 250.395,A -85,B 0,C 180,E1 -16012.074,E2 -16012.074} C_VEL
LIN {X 0,Y 305.69,Z 250.405,A -85,B 0,C 180,E1 -16014.724,E2 -16014.724} C_VEL
LIN {X 0,Y 305.962,Z 250.371,A -85,B 0,C 180,E1 -16018.684,E2 -16018.684} C_VEL
LIN {X 0,Y 305.956,Z 250.373,A -85,B 0,C 180,E1 -16021.316,E2 -16021.316} C_VEL
LIN {X 0,Y 305.791,Z 250.392,A -85,B 0,C 180,E1 -16026.599,E2 -16026.599} C_VEL
LIN {X 0,Y 305.703,Z 250.406,A -85,B 0,C 180,E1 -16029.261,E2 -16029.261} C_VEL
LIN {X 0,Y 305.595,Z 250.419,A -85,B 0,C 180,E1 -16033.296,E2 -16033.296} C_VEL
LIN {X 0,Y 305.56,Z 250.42,A -85,B 0,C 180,E1 -16036.022,E2 -16036.022} C_VEL
LIN {X 0,Y 305.55,Z 250.421,A -85,B 0,C 180,E1 -16039.426,E2 -16039.426} C_VEL
LIN {X 0,Y 305.464,Z 250.435,A -85,B 0,C 180,E1 -16043.025,E2 -16043.025} C_VEL
LIN {X 0,Y 305.459,Z 250.434,A -85,B 0,C 180,E1 -16046.189,E2 -16046.189} C_VEL
LIN {X 0,Y 305.443,Z 250.436,A -85,B 0,C 180,E1 -16049.028,E2 -16049.028} C_VEL
LIN {X 0,Y 305.444,Z 250.436,A -85,B 0,C 180,E1 -16051.952,E2 -16051.952} C_VEL
LIN {X 0,Y 305.47,Z 250.433,A -85,B 0,C 180,E1 -16055.113,E2 -16055.113} C_VEL
LIN {X 0,Y 305.457,Z 250.437,A -85,B 0,C 180,E1 -16058.528,E2 -16058.528} C_VEL
LIN {X 0,Y 305.462,Z 250.435,A -85,B 0,C 180,E1 -16062.585,E2 -16062.585} C_VEL
LIN {X 0,Y 305.428,Z 250.441,A -85,B 0,C 180,E1 -16066.343,E2 -16066.343} C_VEL
LIN {X 0,Y 305.416,Z 250.443,A -85,B 0,C 180,E1 -16069.884,E2 -16069.884} C_VEL
LIN {X 0,Y 305.468,Z 250.435,A -85,B 0,C 180,E1 -16073.636,E2 -16073.636} C_VEL
LIN {X 0,Y 305.446,Z 250.435,A -85,B 0,C 180,E1 -16076.479,E2 -16076.479} C_VEL
LIN {X 0,Y 305.221,Z 250.464,A -85,B 0,C 180,E1 -16079.562,E2 -16079.562} C_VEL
LIN {X 0,Y 304.925,Z 250.727,A -85,B 0,C 180,E1 -16082.549,E2 -16082.549} C_VEL
LIN {X 0,Y 304.823,Z 253.088,A -85,B 0,C 180,E1 -16085.478,E2 -16085.478} C_VEL
LIN {X 0,Y 304.68,Z 255.5,A -85,B 0,C 180,E1 -16088.34,E2 -16088.34} C_VEL
LIN {X 0,Y 304.619,Z 257.801,A -85,B 0,C 180,E1 -16090.995,E2 -16090.995} C_VEL
LIN {X 0,Y 308.608,Z 271.234,A -85,B 0,C 180,E1 -16091.92,E2 -16091.92} C_VEL
LIN {X 0,Y 311.514,Z 283.176,A -85,B 0,C 180,E1 -16092.943,E2 -16092.943} C_VEL
LIN {X 0,Y 312.871,Z 290.064,A -85,B 0,C 180,E1 -16093.63,E2 -16093.63} C_VEL
LIN {X 0,Y 312.056,Z 300.362,A -85,B 0,C 180,E1 -16094.653,E2 -16094.653} C_VEL
LIN {X 0,Y 310.872,Z 310.756,A -85,B 0,C 180,E1 -16095.933,E2 -16095.933} C_VEL
LIN {X 0,Y 309.552,Z 320.635,A -85,B 0,C 180,E1 -16097.438,E2 -16097.438} C_VEL
LIN {X 0,Y 308.171,Z 329.958,A -85,B 0,C 180,E1 -16099.198,E2 -16099.198} C_VEL
LIN {X 0,Y 307.124,Z 337.993,A -85,B 0,C 180,E1 -16101.113,E2 -16101.113} C_VEL
LIN {X 0,Y 306.204,Z 343.656,A -85,B 0,C 180,E1 -16102.746,E2 -16102.746} C_VEL
LIN {X 0,Y 305.288,Z 349.177,A -85,B 0,C 180,E1 -16104.715,E2 -16104.715} C_VEL
LIN {X 0,Y 304.645,Z 353.519,A -85,B 0,C 180,E1 -16106.692,E2 -16106.692} C_VEL
LIN {X 0,Y 304.25,Z 356.804,A -85,B 0,C 180,E1 -16108.674,E2 -16108.674} C_VEL
LIN {X 0,Y 304.133,Z 358.435,A -85,B 0,C 180,E1 -16109.998,E2 -16109.998} C_VEL
LIN {X 0,Y 304.046,Z 359.674,A -85,B 0,C 180,E1 -16111.323,E2 -16111.323} C_VEL
LIN {X 0,Y 303.945,Z 360.527,A -85,B 0,C 180,E1 -16112.649,E2 -16112.649} C_VEL
LIN {X 0,Y 304.039,Z 360.988,A -85,B 0,C 180,E1 -16115.303,E2 -16115.303} C_VEL
LIN {X 0,Y 304.246,Z 359.937,A -85,B 0,C 180,E1 -16117.965,E2 -16117.965} C_VEL
LIN {X 0,Y 304.416,Z 358.783,A -85,B 0,C 180,E1 -16119.298,E2 -16119.298} C_VEL
LIN {X 0,Y 304.719,Z 357.221,A -85,B 0,C 180,E1 -16120.631,E2 -16120.631} C_VEL
LIN {X 0,Y 305.322,Z 354.071,A -85,B 0,C 180,E1 -16122.629,E2 -16122.629} C_VEL
LIN {X 0,Y 306.364,Z 348.796,A -85,B 0,C 180,E1 -16125.062,E2 -16125.062} C_VEL
LIN {X 0,Y 307.674,Z 342.338,A -85,B 0,C 180,E1 -16127.272,E2 -16127.272} C_VEL
LIN {X 0,Y 309.138,Z 335.004,A -85,B 0,C 180,E1 -16129.245,E2 -16129.245} C_VEL
LIN {X 0,Y 310.826,Z 325.853,A -85,B 0,C 180,E1 -16131.207,E2 -16131.207} C_VEL
LIN {X 0,Y 312.406,Z 316.307,A -85,B 0,C 180,E1 -16132.831,E2 -16132.831} C_VEL
LIN {X 0,Y 314.05,Z 305.671,A -85,B 0,C 180,E1 -16134.278,E2 -16134.278} C_VEL
LIN {X 0,Y 315.421,Z 295.248,A -85,B 0,C 180,E1 -16135.41,E2 -16135.41} C_VEL
LIN {X 0,Y 313.163,Z 283.968,A -85,B 0,C 180,E1 -16136.667,E2 -16136.667} C_VEL
LIN {X 0,Y 309.628,Z 271.636,A -85,B 0,C 180,E1 -16137.855,E2 -16137.855} C_VEL
LIN {X 0,Y 305.666,Z 260.798,A -85,B 0,C 180,E1 -16138.766,E2 -16138.766} C_VEL
LIN {X 0,Y 304.884,Z 258.266,A -85,B 0,C 180,E1 -16138.95,E2 -16138.95} C_VEL
LIN {X 0,Y 305.056,Z 255.779,A -85,B 0,C 180,E1 -16141.995,E2 -16141.995} C_VEL
LIN {X 0,Y 305.169,Z 253.276,A -85,B 0,C 180,E1 -16145.149,E2 -16145.149} C_VEL
LIN {X 0,Y 305.316,Z 250.787,A -85,B 0,C 180,E1 -16148.497,E2 -16148.497} C_VEL
LIN {X 0,Y 305.378,Z 250.445,A -85,B 0,C 180,E1 -16150.582,E2 -16150.582} C_VEL
LIN {X 0,Y 305.414,Z 250.442,A -85,B 0,C 180,E1 -16153.654,E2 -16153.654} C_VEL
LIN {X 0,Y 305.447,Z 250.438,A -85,B 0,C 180,E1 -16157.412,E2 -16157.412} C_VEL
LIN {X 0,Y 305.487,Z 250.432,A -85,B 0,C 180,E1 -16161.599,E2 -16161.599} C_VEL
LIN {X 0,Y 305.454,Z 250.437,A -85,B 0,C 180,E1 -16164.885,E2 -16164.885} C_VEL
LIN {X 0,Y 305.44,Z 250.437,A -85,B 0,C 180,E1 -16168.354,E2 -16168.354} C_VEL
LIN {X 0,Y 305.504,Z 250.431,A -85,B 0,C 180,E1 -16171.112,E2 -16171.112} C_VEL
LIN {X 0,Y 305.561,Z 250.424,A -85,B 0,C 180,E1 -16174.087,E2 -16174.087} C_VEL
LIN {X 0,Y 305.491,Z 250.432,A -85,B 0,C 180,E1 -16178.402,E2 -16178.402} C_VEL
LIN {X 0,Y 305.58,Z 250.42,A -85,B 0,C 180,E1 -16181.217,E2 -16181.217} C_VEL
LIN {X 0,Y 305.638,Z 250.415,A -85,B 0,C 180,E1 -16185.348,E2 -16185.348} C_VEL
LIN {X 0,Y 305.605,Z 250.416,A -85,B 0,C 180,E1 -16185.715,E2 -16185.715} C_VEL
LIN {X 0,Y 304.908,Z 250.504,A -85,B 0,C 180,E1 -16186.814,E2 -16186.814} C_VEL
LIN {X 0,Y 302.125,Z 250.851,A -85,B 0,C 180,E1 -16188.607,E2 -16188.607} C_VEL
LIN {X 0,Y 299.803,Z 251.141,A -85,B 0,C 180,E1 -16190.061,E2 -16190.061} C_VEL
LIN {X 0,Y 298.819,Z 251.263,A -85,B 0,C 180,E1 -16191.185,E2 -16191.185} C_VEL
LIN {X 0,Y 298.744,Z 251.272,A -85,B 0,C 180,E1 -16191.565,E2 -16191.565} C_VEL
LIN {X 0,Y 298.654,Z 251.284,A -85,B 0,C 180,E1 -16194.599,E2 -16194.599} C_VEL
LIN {X 0,Y 298.913,Z 251.252,A -85,B 0,C 180,E1 -16198.653,E2 -16198.653} C_VEL
LIN {X 0,Y 298.911,Z 251.252,A -85,B 0,C 180,E1 -16201.347,E2 -16201.347} C_VEL
LIN {X 0,Y 298.789,Z 251.266,A -85,B 0,C 180,E1 -16206.754,E2 -16206.754} C_VEL
LIN {X 0,Y 298.669,Z 251.281,A -85,B 0,C 180,E1 -16209.481,E2 -16209.481} C_VEL
LIN {X 0,Y 298.541,Z 251.298,A -85,B 0,C 180,E1 -16213.616,E2 -16213.616} C_VEL
LIN {X 0,Y 298.538,Z 251.294,A -85,B 0,C 180,E1 -16216.409,E2 -16216.409} C_VEL
LIN {X 0,Y 298.501,Z 251.299,A -85,B 0,C 180,E1 -16219.656,E2 -16219.656} C_VEL
LIN {X 0,Y 298.447,Z 251.312,A -85,B 0,C 180,E1 -16223.598,E2 -16223.598} C_VEL
LIN {X 0,Y 298.479,Z 251.307,A -85,B 0,C 180,E1 -16226.575,E2 -16226.575} C_VEL
LIN {X 0,Y 298.416,Z 251.314,A -85,B 0,C 180,E1 -16229.642,E2 -16229.642} C_VEL
LIN {X 0,Y 298.388,Z 251.317,A -85,B 0,C 180,E1 -16232.801,E2 -16232.801} C_VEL
LIN {X 0,Y 298.437,Z 251.31,A -85,B 0,C 180,E1 -16236.809,E2 -16236.809} C_VEL
LIN {X 0,Y 298.482,Z 251.597,A -85,B 0,C 180,E1 -16237.748,E2 -16237.748} C_VEL
LIN {X 0,Y 299.112,Z 255.402,A -85,B 0,C 180,E1 -16241.25,E2 -16241.25} C_VEL
LIN {X 0,Y 299.876,Z 259.378,A -85,B 0,C 180,E1 -16244.676,E2 -16244.676} C_VEL
LIN {X 0,Y 300.73,Z 264.08,A -85,B 0,C 180,E1 -16248.403,E2 -16248.403} C_VEL
LIN {X 0,Y 301.46,Z 268.642,A -85,B 0,C 180,E1 -16251.769,E2 -16251.769} C_VEL
LIN {X 0,Y 301.504,Z 271.197,A -85,B 0,C 180,E1 -16253.533,E2 -16253.533} C_VEL
LIN {X 0,Y 300.666,Z 276.031,A -85,B 0,C 180,E1 -16256.684,E2 -16256.684} C_VEL
LIN {X 0,Y 299.467,Z 283.299,A -85,B 0,C 180,E1 -16261.245,E2 -16261.245} C_VEL
LIN {X 0,Y 298.644,Z 288.978,A -85,B 0,C 180,E1 -16264.737,E2 -16264.737} C_VEL
LIN {X 0,Y 300.58,Z 297.308,A -85,B 0,C 180,E1 -16265.249,E2 -16265.249} C_VEL
LIN {X 0,Y 303.02,Z 308.96,A -85,B 0,C 180,E1 -16266.133,E2 -16266.133} C_VEL
LIN {X 0,Y 304.741,Z 321.811,A -85,B 0,C 180,E1 -16267.293,E2 -16267.293} C_VEL
LIN {X 0,Y 305.389,Z 333.741,A -85,B 0,C 180,E1 -16268.574,E2 -16268.574} C_VEL
LIN {X 0,Y 305.429,Z 339.476,A -85,B 0,C 180,E1 -16269.283,E2 -16269.283} C_VEL
LIN {X 0,Y 303.617,Z 350.285,A -85,B 0,C 180,E1 -16270.742,E2 -16270.742} C_VEL
LIN {X 0,Y 301.934,Z 360.027,A -85,B 0,C 180,E1 -16272.389,E2 -16272.389} C_VEL
LIN {X 0,Y 300.59,Z 368.035,A -85,B 0,C 180,E1 -16274.057,E2 -16274.057} C_VEL
LIN {X 0,Y 299.206,Z 375.906,A -85,B 0,C 180,E1 -16276.071,E2 -16276.071} C_VEL
LIN {X 0,Y 297.932,Z 383.131,A -85,B 0,C 180,E1 -16278.435,E2 -16278.435} C_VEL
LIN {X 0,Y 297.272,Z 387.982,A -85,B 0,C 180,E1 -16280.476,E2 -16280.476} C_VEL
LIN {X 0,Y 296.853,Z 391.721,A -85,B 0,C 180,E1 -16282.52,E2 -16282.52} C_VEL
LIN {X 0,Y 296.688,Z 394.45,A -85,B 0,C 180,E1 -16284.565,E2 -16284.565} C_VEL
LIN {X 0,Y 296.663,Z 395.747,A -85,B 0,C 180,E1 -16285.927,E2 -16285.927} C_VEL
LIN {X 0,Y 296.622,Z 396.641,A -85,B 0,C 180,E1 -16287.286,E2 -16287.286} C_VEL
LIN {X 0,Y 296.663,Z 397.098,A -85,B 0,C 180,E1 -16288.645,E2 -16288.645} C_VEL
LIN {X 0,Y 296.782,Z 397.161,A -85,B 0,C 180,E1 -16290.002,E2 -16290.002} C_VEL
LIN {X 0,Y 296.699,Z 396.82,A -85,B 0,C 180,E1 -16291.359,E2 -16291.359} C_VEL
LIN {X 0,Y 296.642,Z 396.086,A -85,B 0,C 180,E1 -16292.718,E2 -16292.718} C_VEL
LIN {X 0,Y 296.691,Z 394.913,A -85,B 0,C 180,E1 -16294.077,E2 -16294.077} C_VEL
LIN {X 0,Y 296.739,Z 392.717,A -85,B 0,C 180,E1 -16295.882,E2 -16295.882} C_VEL
LIN {X 0,Y 296.979,Z 388.802,A -85,B 0,C 180,E1 -16298.165,E2 -16298.165} C_VEL
LIN {X 0,Y 297.455,Z 384.12,A -85,B 0,C 180,E1 -16300.209,E2 -16300.209} C_VEL
LIN {X 0,Y 298.349,Z 377.048,A -85,B 0,C 180,E1 -16302.587,E2 -16302.587} C_VEL
LIN {X 0,Y 299.462,Z 369.403,A -85,B 0,C 180,E1 -16304.615,E2 -16304.615} C_VEL
LIN {X 0,Y 300.654,Z 361.595,A -85,B 0,C 180,E1 -16306.292,E2 -16306.292} C_VEL
LIN {X 0,Y 301.948,Z 352.052,A -85,B 0,C 180,E1 -16307.965,E2 -16307.965} C_VEL
LIN {X 0,Y 303.467,Z 341.481,A -85,B 0,C 180,E1 -16309.447,E2 -16309.447} C_VEL
LIN {X 0,Y 304.091,Z 335.934,A -85,B 0,C 180,E1 -16310.109,E2 -16310.109} C_VEL
LIN {X 0,Y 303.266,Z 324.182,A -85,B 0,C 180,E1 -16311.399,E2 -16311.399} C_VEL
LIN {X 0,Y 301.986,Z 311.488,A -85,B 0,C 180,E1 -16312.502,E2 -16312.502} C_VEL
LIN {X 0,Y 299.998,Z 298.516,A -85,B 0,C 180,E1 -16313.393,E2 -16313.393} C_VEL
LIN {X 0,Y 298.241,Z 289.265,A -85,B 0,C 180,E1 -16313.894,E2 -16313.894} C_VEL
LIN {X 0,Y 299.081,Z 282.396,A -85,B 0,C 180,E1 -16318.035,E2 -16318.035} C_VEL
LIN {X 0,Y 299.987,Z 276.159,A -85,B 0,C 180,E1 -16321.81,E2 -16321.81} C_VEL
LIN {X 0,Y 300.878,Z 270.795,A -85,B 0,C 180,E1 -16325.16,E2 -16325.16} C_VEL
LIN {X 0,Y 301.111,Z 267.167,A -85,B 0,C 180,E1 -16327.48,E2 -16327.48} C_VEL
LIN {X 0,Y 300.733,Z 264.154,A -85,B 0,C 180,E1 -16329.539,E2 -16329.539} C_VEL
LIN {X 0,Y 299.793,Z 258.854,A -85,B 0,C 180,E1 -16333.387,E2 -16333.387} C_VEL
LIN {X 0,Y 298.914,Z 254.232,A -85,B 0,C 180,E1 -16337.012,E2 -16337.012} C_VEL
LIN {X 0,Y 298.419,Z 251.315,A -85,B 0,C 180,E1 -16339.49,E2 -16339.49} C_VEL
LIN {X 0,Y 298.451,Z 251.309,A -85,B 0,C 180,E1 -16343.194,E2 -16343.194} C_VEL
LIN {X 0,Y 298.4,Z 251.314,A -85,B 0,C 180,E1 -16347.2,E2 -16347.2} C_VEL
LIN {X 0,Y 298.417,Z 251.313,A -85,B 0,C 180,E1 -16350.623,E2 -16350.623} C_VEL
LIN {X 0,Y 298.458,Z 251.306,A -85,B 0,C 180,E1 -16354.922,E2 -16354.922} C_VEL
LIN {X 0,Y 298.423,Z 251.312,A -85,B 0,C 180,E1 -16357.864,E2 -16357.864} C_VEL
LIN {X 0,Y 298.485,Z 251.303,A -85,B 0,C 180,E1 -16360.753,E2 -16360.753} C_VEL
LIN {X 0,Y 298.519,Z 251.298,A -85,B 0,C 180,E1 -16364.991,E2 -16364.991} C_VEL
LIN {X 0,Y 298.589,Z 251.29,A -85,B 0,C 180,E1 -16369.147,E2 -16369.147} C_VEL
LIN {X 0,Y 298.726,Z 251.275,A -85,B 0,C 180,E1 -16371.885,E2 -16371.885} C_VEL
LIN {X 0,Y 298.66,Z 251.281,A -85,B 0,C 180,E1 -16374.599,E2 -16374.599} C_VEL
LIN {X 0,Y 298.929,Z 251.247,A -85,B 0,C 180,E1 -16378.653,E2 -16378.653} C_VEL
LIN {X 0,Y 298.923,Z 251.25,A -85,B 0,C 180,E1 -16381.347,E2 -16381.347} C_VEL
LIN {X 0,Y 298.74,Z 251.271,A -85,B 0,C 180,E1 -16386.755,E2 -16386.755} C_VEL
LIN {X 0,Y 298.634,Z 251.285,A -85,B 0,C 180,E1 -16389.482,E2 -16389.482} C_VEL
LIN {X 0,Y 298.554,Z 251.293,A -85,B 0,C 180,E1 -16393.616,E2 -16393.616} C_VEL
